(* IEC 61131-3 sources: Elmo_Master/Lasal_PRG/Elmo_EtherCAT_Test_4Axis/Class/LMCDiagnosticsService (part 2) *)

	if detailCode <> 0 then
		(pResponse + 12)^$UDINT := detailCode;
		RETURN;
	end_if;
	if ResponseCapacity < 156 then
		ResponseSize := -1;
		RETURN;
	end_if;

	_memset(dest:=pResponse, usByte:=0, cntr:=156);
	pResponse^$UINT := LMC_DIAG_SCHEMA_VERSION;
	(pResponse + 4)^$UINT := 0;
	(pResponse + 6)^$INT := 0;
	(pResponse + 8)^$UDINT := requestId;
	(pResponse + 12)^$UDINT := 0;
	(pResponse + 16)^$UINT := baseState$UINT;
	(pResponse + 18)^$UINT := EncoderMaintenanceState[recordBase + 1]$UINT;
	(pResponse + 20)^$UDINT := EncoderMaintenanceState[recordBase + 2]$UDINT;
	(pResponse + 24)^$UDINT := EncoderMaintenanceState[recordBase + 3]$UDINT;
	(pResponse + 28)^$UDINT := EncoderMaintenanceState[recordBase + 4]$UDINT;
	(pResponse + 32)^$UDINT := EncoderMaintenanceState[recordBase + 5]$UDINT;
	(pResponse + 36)^$UDINT := EncoderMaintenanceState[recordBase + 6]$UDINT;
	(pResponse + 40)^$UDINT := EncoderMaintenanceState[recordBase + 7]$UDINT;
	(pResponse + 44)^$UDINT := EncoderMaintenanceState[recordBase + 8]$UDINT;
	(pResponse + 48)^$UDINT := EncoderMaintenanceState[recordBase + 9]$UDINT;
	(pResponse + 52)^$UINT := EncoderMaintenanceState[recordBase + 10]$UINT;
	(pResponse + 54)^$UINT := EncoderMaintenanceState[recordBase + 11]$UINT;
	(pResponse + 56)^$UINT := EncoderMaintenanceState[recordBase + 12]$UINT;
	(pResponse + 58)^$UINT := 0;
	(pResponse + 60)^$UDINT := EncoderMaintenanceState[recordBase + 13]$UDINT;
	(pResponse + 64)^$UDINT := EncoderMaintenanceState[recordBase + 14]$UDINT;
	(pResponse + 68)^$UDINT := EncoderMaintenanceState[recordBase + 15]$UDINT;
	(pResponse + 72)^$UDINT := EncoderMaintenanceState[recordBase + 16]$UDINT;
	(pResponse + 76)^$UDINT := EncoderMaintenanceState[recordBase + 17]$UDINT;
	(pResponse + 80)^$UDINT := EncoderMaintenanceState[recordBase + 18]$UDINT;
	(pResponse + 84)^$UINT := EncoderMaintenanceState[recordBase + 19]$UINT;
	(pResponse + 86)^$INT := EncoderMaintenanceState[recordBase + 20]$INT;
	(pResponse + 88)^$UDINT := EncoderMaintenanceState[recordBase + 21]$UDINT;
	(pResponse + 92)^$UDINT := EncoderMaintenanceState[recordBase + 22]$UDINT;
	(pResponse + 96)^$UDINT := EncoderMaintenanceState[recordBase + 23]$UDINT;
	(pResponse + 100)^$UDINT := EncoderMaintenanceState[recordBase + 24]$UDINT;
	(pResponse + 104)^$UDINT := EncoderMaintenanceState[recordBase + 25]$UDINT;
	(pResponse + 108)^$UDINT := EncoderMaintenanceState[recordBase + 26]$UDINT;
	(pResponse + 112)^$UDINT := EncoderMaintenanceState[recordBase + 27]$UDINT;
	(pResponse + 116)^$UDINT := EncoderMaintenanceState[recordBase + 28]$UDINT;
	(pResponse + 120)^$UDINT := EncoderMaintenanceState[recordBase + 29]$UDINT;
	(pResponse + 124)^$UDINT := EncoderMaintenanceState[recordBase + 30]$UDINT;
	(pResponse + 128)^$UDINT := EncoderMaintenanceState[recordBase + 31]$UDINT;
	(pResponse + 132)^$UINT := EncoderMaintenanceState[recordBase + 32]$UINT;
	(pResponse + 134)^$UINT := 0;
	(pResponse + 136)^$DINT := EncoderMaintenanceState[recordBase + 33];
	(pResponse + 140)^$UDINT := EncoderMaintenanceState[recordBase + 34]$UDINT;
	(pResponse + 144)^$DINT := EncoderMaintenanceState[recordBase + 35];
	(pResponse + 148)^$UDINT := EncoderMaintenanceState[recordBase + 36]$UDINT;
	(pResponse + 152)^$UDINT := EncoderMaintenanceState[recordBase + 37]$UDINT;
	ResponseSize := 156;

END_FUNCTION

FUNCTION LMCDiagnosticsService::HandleEncoderMaintenanceRetire
	VAR_INPUT
		Reference 	: UINT;
		pRequest 	: ^USINT;
		pResponse 	: ^USINT;
		ResponseCapacity 	: UDINT;
		CallerSessionEpoch 	: UDINT;
		RequestSize 	: UDINT;
	END_VAR
	VAR_OUTPUT
		ResponseSize 	: DINT;
	END_VAR
	VAR
		driveReference : UINT;
		requestId, recordGeneration, detailCode : UDINT;
		rawState, baseState : UDINT;
		recordBase : DINT;
		stateValid : BOOL;
	END_VAR

	ResponseSize := -1;
	if (pResponse = NIL) | (ResponseCapacity < 16) then
		RETURN;
	end_if;
	_memset(dest:=pResponse, usByte:=0, cntr:=16);
	pResponse^$UINT := LMC_DIAG_SCHEMA_VERSION;
	(pResponse + 4)^$UINT := 1;
	(pResponse + 6)^$INT := LMC_DIAG_ERROR_ID;
	requestId := 0;
	if (pRequest <> NIL) & (RequestSize >= 8) then
		requestId := (pRequest + 4)^$UDINT;
	end_if;
	(pResponse + 8)^$UDINT := requestId;
	ResponseSize := 16;
	detailCode := LMC_DIAG_ENCODER_DETAIL_KEY_MISMATCH;

	if (pRequest = NIL) | (RequestSize <> 76) | (Reference <> 0) then
		(pResponse + 12)^$UDINT := detailCode;
		RETURN;
	end_if;
	driveReference := (pRequest + 44)^$UINT;
	recordGeneration := (pRequest + 72)^$UDINT;
	recordBase := 0;
	if (driveReference < 1) | (driveReference > 4) |
		(recordGeneration = 0) then
		(pResponse + 12)^$UDINT := detailCode;
		RETURN;
	end_if;

	recordBase := TO_DINT(driveReference - 1) *
		LMC_DIAG_ENCODER_RECORD_STRIDE;
	rawState := EncoderMaintenanceState[recordBase]$UDINT;
	baseState := rawState and 0x00007FFF;
	stateValid :=
		(rawState = LMC_DIAG_ENCODER_RECORD_SUCCEEDED) |
		(rawState = LMC_DIAG_ENCODER_RECORD_FAILED) |
		(rawState = LMC_DIAG_ENCODER_RECORD_ABORTED) |
		(rawState = (LMC_DIAG_ENCODER_RECORD_RETIRED OR
		 LMC_DIAG_ENCODER_RECORD_SUCCEEDED)) |
		(rawState = (LMC_DIAG_ENCODER_RECORD_RETIRED OR
		 LMC_DIAG_ENCODER_RECORD_FAILED)) |
		(rawState = (LMC_DIAG_ENCODER_RECORD_RETIRED OR
		 LMC_DIAG_ENCODER_RECORD_ABORTED));
	if rawState = 0 then
		detailCode := LMC_DIAG_ENCODER_DETAIL_NOT_FOUND;
	elsif rawState = LMC_DIAG_ENCODER_RECORD_RUNNING then
		detailCode := LMC_DIAG_ENCODER_DETAIL_INDETERMINATE;
	elsif stateValid = FALSE then
		detailCode := LMC_DIAG_ENCODER_DETAIL_STORE_CORRUPT;
	elsif EncoderMaintenanceState[recordBase + 36]$UDINT <>
		recordGeneration then
		detailCode := LMC_DIAG_ENCODER_DETAIL_KEY_MISMATCH;
	else
		ResponseSize := HandleEncoderMaintenanceOutcome(
			Reference:=Reference, pRequest:=pRequest,
			pResponse:=pResponse, ResponseCapacity:=ResponseCapacity,
			CallerSessionEpoch:=CallerSessionEpoch, RequestSize:=72);
		if (ResponseSize = 156) &
			((pResponse + 148)^$UDINT = recordGeneration) then
			if rawState = baseState then
				// State is the publication word. Setting the tombstone last makes
				// retrying the same exact retirement idempotent.
				EncoderMaintenanceState[recordBase] :=
					TO_DINT(baseState OR
					LMC_DIAG_ENCODER_RECORD_RETIRED);
			end_if;
			RETURN;
		end_if;
		detailCode := LMC_DIAG_ENCODER_DETAIL_KEY_MISMATCH;
	end_if;

	(pResponse + 4)^$UINT := 1;
	(pResponse + 6)^$INT := LMC_DIAG_ERROR_ID;
	(pResponse + 12)^$UDINT := detailCode;
	ResponseSize := 16;

END_FUNCTION

FUNCTION LMCDiagnosticsService::ProcessEncoderMaintenance
	VAR
		snapshot : ARRAY [0..303] OF USINT;
		preemptionSnapshot : ARRAY [0..215] OF USINT;
		completion : LMCSdoExecutor::LMCSdoExecutorResult;
		stage, recordBase, desiredTerminalState : DINT;
		axisReference, maintenanceObjectIndex : UINT;
		maintenanceSubIndex : USINT;
		maintenanceKind, preemptionCleanupKind : UINT;
		maintenanceWriteValue : UINT;
		axisMask, encoderProcessOperationToken, admissionToken, ownerGeneration : UDINT;
		callerSessionEpoch, requestSequence : UDINT;
		maintenanceCommandValue, timeoutMilliseconds : UDINT;
		expectedExecuteToken, safetyAdmissionToken, safetyOwnerGeneration : UDINT;
		serviceNow, serviceStartMs, cleanupStartMs : UDINT;
		elapsedMs, remainingMs, currentCycle, previousCycle : UDINT;
		healthOffset, valueOffset, controlWord, statusWord : UDINT;
		failureDetail, failureNative, verificationFlags : UDINT;
		axisError, actualPosition : DINT;
		copyResult, ownerResult, orphanResult, preemptionResult : DINT;
		startResult : iprStates;
		snapshotValid, newCycle, motorOff : BOOL;
		executorConnected, executorReusable, featureEnabled : BOOL;
		safeFailure, quarantine, preemptionSnapshotValid : BOOL;
		dispatchDefinitelyAbsent, publishPreemptionCleanup : BOOL;
	END_VAR

	stage := EncoderMaintenanceState[LMC_DIAG_ENCODER_RUNTIME_BASE];
	if stage = LMC_DIAG_ENCODER_STAGE_IDLE then
		RETURN;
	end_if;

	recordBase := EncoderMaintenanceState[154];
	axisReference := EncoderMaintenanceState[153]$UINT;
	admissionToken := EncoderMaintenanceState[160]$UDINT;
	ownerGeneration := EncoderMaintenanceState[161]$UDINT;
	_memset(dest:=#preemptionSnapshot[0], usByte:=0,
		cntr:=sizeof(preemptionSnapshot));
	preemptionResult := -1;
	if IsClientConnected(#AxisOwnership) & (admissionToken <> 0) &
		(ownerGeneration <> 0) then
		preemptionResult := AxisOwnership.CopyAxisOwnershipPreemption(
			PreemptedAdmissionToken:=admissionToken,
			PreemptedOwnerGeneration:=ownerGeneration,
			pDest:=#preemptionSnapshot[0],
			DestSize:=sizeof(preemptionSnapshot));
	end_if;
	if preemptionResult = LMC_DIAG_PREEMPT_PENDING_FREEZE then
		// Safety is only reserved. Freeze before changing any owner runtime word.
		RETURN;
	end_if;
	if (preemptionResult < 0) |
		(preemptionResult > LMC_DIAG_PREEMPT_CLEANUP_QUARANTINED) then
		EncoderMaintenanceState[179] :=
			LMC_DIAG_ENCODER_DETAIL_STORE_CORRUPT;
		EncoderMaintenanceState[180] := TO_DINT(0 - preemptionResult);
		EncoderMaintenanceState[152] :=
			LMC_DIAG_ENCODER_STAGE_QUARANTINED;
		RETURN;
	end_if;
	if (sizeof(EncoderMaintenanceState) <> 768) |
		(axisReference < 1) | (axisReference > 4) |
		(recordBase <> (TO_DINT(axisReference - 1) *
		 LMC_DIAG_ENCODER_RECORD_STRIDE)) |
		(EncoderMaintenanceState[recordBase] <>
		 LMC_DIAG_ENCODER_RECORD_RUNNING) then
		EncoderMaintenanceState[152] :=
			LMC_DIAG_ENCODER_STAGE_QUARANTINED;
		RETURN;
	end_if;

	axisMask := TO_UDINT(1) shl TO_UDINT(axisReference - 1);
	maintenanceKind := EncoderMaintenanceState[182]$UINT;
	maintenanceObjectIndex := EncoderMaintenanceState[157]$UINT;
	maintenanceSubIndex := EncoderMaintenanceState[158]$USINT;
	maintenanceCommandValue := EncoderMaintenanceState[159]$UDINT;
	maintenanceWriteValue := LMC_DIAG_ENCODER_RESET_VALUE;
	timeoutMilliseconds := EncoderMaintenanceState[recordBase + 14]$UDINT;
	encoderProcessOperationToken := EncoderMaintenanceState[155]$UDINT;
	callerSessionEpoch := EncoderMaintenanceState[162]$UDINT;
	requestSequence := EncoderMaintenanceState[163]$UDINT;
	serviceNow := ops.tAbsolute;
	serviceStartMs := EncoderMaintenanceState[164]$UDINT;
	cleanupStartMs := EncoderMaintenanceState[165]$UDINT;
	elapsedMs := serviceNow - serviceStartMs;
	previousCycle := EncoderMaintenanceState[166]$UDINT;
	currentCycle := previousCycle;
	controlWord := EncoderMaintenanceState[168]$UDINT;
	statusWord := EncoderMaintenanceState[169]$UDINT;
	axisError := EncoderMaintenanceState[170];
	actualPosition := EncoderMaintenanceState[171];
	expectedExecuteToken := 0;
	if maintenanceKind = 1 then
		expectedExecuteToken := 0x30325754;
	elsif maintenanceKind = 2 then
		expectedExecuteToken := 0x39315754;
	end_if;

	preemptionResult := HandleEncoderMaintenancePreemption(
		Stage:=stage,
		PreemptionResult:=preemptionResult,
		pPreemptionSnapshot:=#preemptionSnapshot[0],
		ServiceNow:=serviceNow);
	if preemptionResult <> 0 then
		RETURN;
	end_if;

	if stage = LMC_DIAG_ENCODER_STAGE_QUARANTINED then
		RETURN;
	end_if;
	EncoderMaintenanceServiceMilliseconds := serviceNow;

	snapshotValid := FALSE;
	newCycle := FALSE;
	motorOff := FALSE;
	copyResult := -1;
	if IsClientConnected(#InputLatch) then
		copyResult := InputLatch.CopySnapshot(
			pDest:=#snapshot[0], DestSize:=sizeof(snapshot));
	end_if;
	if (copyResult = 0) & (snapshot[0]$UDINT <> 0) then
		currentCycle := snapshot[0]$UDINT;
		healthOffset := 64 + TO_UDINT(axisReference - 1) * 36;
		valueOffset := 208 + TO_UDINT(axisReference - 1) * 24;
		controlWord := snapshot[TO_DINT(valueOffset + 8)]$UDINT;
		statusWord := snapshot[TO_DINT(valueOffset + 20)]$UDINT;
		axisError := snapshot[TO_DINT(healthOffset + 24)]$DINT;
		actualPosition := snapshot[TO_DINT(valueOffset + 12)]$DINT;
		snapshotValid :=
			(snapshot[12]$UDINT = 8) & (snapshot[16]$UDINT = 0) &
			((snapshot[40]$UDINT and 3) = 1) &
			(snapshot[TO_DINT(healthOffset)]$DINT <> 0) &
			(snapshot[TO_DINT(healthOffset + 4)]$UDINT = 8) &
			(snapshot[TO_DINT(healthOffset + 12)]$UDINT = 0) &
			(snapshot[TO_DINT(healthOffset + 16)]$UDINT <>
			 0xFFFFFFFF) &
			(snapshot[TO_DINT(healthOffset + 28)]$UDINT = currentCycle);
		newCycle := snapshotValid & (currentCycle <> previousCycle);
		motorOff := snapshotValid &
			((controlWord and 0x00000008) = 0) &
			((statusWord and 0x00000004) = 0);
		if snapshotValid then
			EncoderMaintenanceState[166] := currentCycle$DINT;
			EncoderMaintenanceState[168] := controlWord$DINT;
			EncoderMaintenanceState[169] := statusWord$DINT;
			EncoderMaintenanceState[170] := axisError;
			EncoderMaintenanceState[171] := actualPosition;
			EncoderMaintenanceState[recordBase + 32] := statusWord$DINT;
			EncoderMaintenanceState[recordBase + 33] := axisError;
			EncoderMaintenanceState[recordBase + 35] := actualPosition;
		end_if;
	end_if;

	executorConnected := FALSE;
	executorReusable := FALSE;
	case axisReference of
		1:
			executorConnected := IsClientConnected(#SdoAxis1) <> 0;
			if executorConnected then
				executorReusable := SdoAxis1.IsReusable();
			end_if;
		2:
			executorConnected := IsClientConnected(#SdoAxis2) <> 0;
			if executorConnected then
				executorReusable := SdoAxis2.IsReusable();
			end_if;
		3:
			executorConnected := IsClientConnected(#SdoAxis3) <> 0;
			if executorConnected then
				executorReusable := SdoAxis3.IsReusable();
			end_if;
		4:
			executorConnected := IsClientConnected(#SdoAxis4) <> 0;
			if executorConnected then
				executorReusable := SdoAxis4.IsReusable();
			end_if;
	end_case;

	featureEnabled :=
		((maintenanceKind = 1) &
		 (LMC_DIAG_ENCODER_TW20_ENABLED = TRUE)) |
		((maintenanceKind = 2) &
		 (LMC_DIAG_ENCODER_TW19_ENABLED = TRUE));
	safeFailure := FALSE;
	quarantine := FALSE;
	failureDetail := LMC_DIAG_ENCODER_DETAIL_EXECUTION;
	failureNative := 0;
	desiredTerminalState := LMC_DIAG_ENCODER_RECORD_FAILED;

	if (maintenanceObjectIndex <> 0x20FC) |
		(((maintenanceKind = 1) & (maintenanceSubIndex <> 0x02)) |
		 ((maintenanceKind = 2) & (maintenanceSubIndex <> 0x01))) |
		((maintenanceKind <> 1) & (maintenanceKind <> 2)) |
		(maintenanceCommandValue <> LMC_DIAG_ENCODER_RESET_VALUE) |
		(encoderProcessOperationToken = 0) | (admissionToken = 0) |
		(ownerGeneration = 0) | (callerSessionEpoch = 0) |
		(requestSequence = 0) | (timeoutMilliseconds < 1) |
		(timeoutMilliseconds > 60000) then
		quarantine := TRUE;
		failureNative := 17;
	elsif (featureEnabled = FALSE) &
		(stage <> LMC_DIAG_ENCODER_STAGE_RELEASE_OWNER) then
		if EncoderMaintenanceState[189]$UDINT = 0 then
			safeFailure := TRUE;
			failureDetail := LMC_DIAG_ENCODER_DETAIL_EXECUTION;
			failureNative := LMC_DIAG_ENCODER_DETAIL_COMPATIBILITY;
		else
			quarantine := TRUE;
			failureNative := LMC_DIAG_ENCODER_DETAIL_COMPATIBILITY;
		end_if;
	end_if;

	if (safeFailure = FALSE) & (quarantine = FALSE) then
		case stage of
			LMC_DIAG_ENCODER_STAGE_PRE_STABLE:
				if elapsedMs >= timeoutMilliseconds then
					safeFailure := TRUE;
					desiredTerminalState :=
						LMC_DIAG_ENCODER_RECORD_ABORTED;
					failureDetail := LMC_DIAG_ENCODER_DETAIL_ABORTED;
				elsif snapshotValid & (motorOff = FALSE) then
					safeFailure := TRUE;
					failureDetail := LMC_DIAG_ENCODER_DETAIL_SEMANTIC;
					failureNative := statusWord;
				elsif newCycle & motorOff then
					EncoderMaintenanceObservedLatchCycle := currentCycle;
					EncoderMaintenanceLatchAdvanceServiceMilliseconds :=
						serviceNow;
					EncoderMaintenanceLatchFreshSampleCount += 1;
					EncoderMaintenanceState[recordBase + 28] :=
						controlWord$DINT;
					EncoderMaintenanceState[recordBase + 30] :=
						statusWord$DINT;
					if EncoderMaintenanceLatchFreshSampleCount >= 3 then
						EncoderMaintenanceState[recordBase + 27]$UDINT :=
							EncoderMaintenanceState[recordBase + 27]$UDINT OR
							LMC_DIAG_ENCODER_VERIFY_MOTOR_OFF_PRE OR
							LMC_DIAG_ENCODER_VERIFY_NO_MOTION;
						EncoderMaintenanceState[152] :=
							LMC_DIAG_ENCODER_STAGE_DISPATCH;
					end_if;
				end_if;

			LMC_DIAG_ENCODER_STAGE_DISPATCH:
				if elapsedMs >= timeoutMilliseconds then
					safeFailure := TRUE;
					desiredTerminalState :=
						LMC_DIAG_ENCODER_RECORD_ABORTED;
					failureDetail := LMC_DIAG_ENCODER_DETAIL_ABORTED;
				elsif snapshotValid = FALSE then
					// Wait only within the same overall service-clock budget.
				elsif motorOff = FALSE then
					safeFailure := TRUE;
					failureDetail := LMC_DIAG_ENCODER_DETAIL_SEMANTIC;
					failureNative := statusWord;
				elsif (executorConnected = FALSE) | (executorReusable = FALSE) |
					(IsClientConnected(#AxisOwnership) = FALSE) then
					quarantine := TRUE;
					failureNative := 24;
				else
					ownerResult := AxisOwnership.ValidateAxisOwnership(
						CommandId:=0x7E53,
						Reference:=axisReference,
						ExpectedAxisMask:=axisMask,
						OwnerKind:=LMC_DIAG_OWNER_KIND_ENCODER,
						ResourceKind:=LMC_DIAG_RESOURCE_DIAGNOSTICS_SDO,
						AdmissionMode:=LMC_DIAG_ADMISSION_LIFECYCLE,
						CallerSessionEpoch:=callerSessionEpoch,
						RequestSequence:=requestSequence,
						AdmissionToken:=admissionToken,
						OwnerGeneration:=ownerGeneration,
						RequiredPhase:=LMC_DIAG_OWNER_PHASE_ACTIVE);
					if ownerResult <> 0 then
						quarantine := TRUE;
						failureNative := TO_UDINT(0 - ownerResult);
					elsif EncoderMaintenanceState[189]$UDINT <> 0 then
						// This is the irreversible one-shot dispatch claim. It is
						// never cleared for retry within an active record.
						quarantine := TRUE;
						failureNative := 25;
					else
						remainingMs := timeoutMilliseconds - elapsedMs;
						if remainingMs < 1 then
							remainingMs := 1;
						end_if;
						if remainingMs > 60000 then
							remainingMs := 60000;
						end_if;
						EncoderMaintenanceState[189]$UDINT := encoderProcessOperationToken;
						startResult := ERROR;
						case axisReference of
							1:
								startResult := SdoAxis1.TryStartWrite(
									OperationToken:=encoderProcessOperationToken,
									ObjectIndex:=maintenanceObjectIndex,
									SubIndex:=maintenanceSubIndex,
									pWriteData:=(#maintenanceWriteValue)$^USINT,
									WriteLength:=2, TimeoutMs:=remainingMs);
							2:
								startResult := SdoAxis2.TryStartWrite(
									OperationToken:=encoderProcessOperationToken,
									ObjectIndex:=maintenanceObjectIndex,
									SubIndex:=maintenanceSubIndex,
									pWriteData:=(#maintenanceWriteValue)$^USINT,
									WriteLength:=2, TimeoutMs:=remainingMs);
							3:
								startResult := SdoAxis3.TryStartWrite(
									OperationToken:=encoderProcessOperationToken,
									ObjectIndex:=maintenanceObjectIndex,
									SubIndex:=maintenanceSubIndex,
									pWriteData:=(#maintenanceWriteValue)$^USINT,
									WriteLength:=2, TimeoutMs:=remainingMs);
							4:
								startResult := SdoAxis4.TryStartWrite(
									OperationToken:=encoderProcessOperationToken,
									ObjectIndex:=maintenanceObjectIndex,
									SubIndex:=maintenanceSubIndex,
									pWriteData:=(#maintenanceWriteValue)$^USINT,
									WriteLength:=2, TimeoutMs:=remainingMs);
						end_case;
						if startResult = READY then
							EncoderMaintenanceState[156] := 1;
							EncoderMaintenanceState[152] :=
								LMC_DIAG_ENCODER_STAGE_WAIT_SDO;
							ownerResult := AxisOwnership.PublishAxisOwnership(
								AxisMask:=axisMask,
								AdmissionToken:=admissionToken,
								OwnerGeneration:=ownerGeneration,
								ReportKind:=LMC_DIAG_OWNER_REPORT_DISPATCH,
								ReportValue0:=TO_UDINT(maintenanceObjectIndex),
								ReportValue1:=encoderProcessOperationToken,
								ObservationCycle:=currentCycle);
							if ownerResult <> 0 then
								// Drain the accepted write before quarantine.
								EncoderMaintenanceState[176] := 1;
							end_if;
						else
							case axisReference of
								1: executorReusable := SdoAxis1.IsReusable();
								2: executorReusable := SdoAxis2.IsReusable();
								3: executorReusable := SdoAxis3.IsReusable();
								4: executorReusable := SdoAxis4.IsReusable();
							end_case;
							if executorReusable then
								safeFailure := TRUE;
								failureNative := TO_UDINT(startResult);
							else
								quarantine := TRUE;
								failureNative := TO_UDINT(startResult);
							end_if;
						end_if;
					end_if;
				end_if;

			LMC_DIAG_ENCODER_STAGE_WAIT_SDO:
				copyResult := -2;
				case axisReference of
					1: copyResult := SdoAxis1.CopyCompletion(
						ExpectedToken:=encoderProcessOperationToken,
						pDest:=#completion, DestSize:=sizeof(completion));
					2: copyResult := SdoAxis2.CopyCompletion(
						ExpectedToken:=encoderProcessOperationToken,
						pDest:=#completion, DestSize:=sizeof(completion));
					3: copyResult := SdoAxis3.CopyCompletion(
						ExpectedToken:=encoderProcessOperationToken,
						pDest:=#completion, DestSize:=sizeof(completion));
					4: copyResult := SdoAxis4.CopyCompletion(
						ExpectedToken:=encoderProcessOperationToken,
						pDest:=#completion, DestSize:=sizeof(completion));
				end_case;
				if copyResult = 0 then
					EncoderMaintenanceState[156] := 0;
					EncoderMaintenanceState[recordBase + 24] :=
						currentCycle$DINT;
					EncoderMaintenanceState[recordBase + 22] :=
						completion.AbortCode$DINT;
					EncoderMaintenanceState[recordBase + 27]$UDINT :=
						EncoderMaintenanceState[recordBase + 27]$UDINT OR
						LMC_DIAG_ENCODER_VERIFY_SDO_COMPLETE OR
						LMC_DIAG_ENCODER_VERIFY_EXECUTOR_DRAINED;
					case axisReference of
						1: executorReusable := SdoAxis1.IsReusable();
						2: executorReusable := SdoAxis2.IsReusable();
						3: executorReusable := SdoAxis3.IsReusable();
						4: executorReusable := SdoAxis4.IsReusable();
					end_case;
					if (completion.Token = encoderProcessOperationToken) &
						(completion.ValidationCode = 0) &
						(completion.OsResult = 0) &
						(completion.AbortCode = 0) &
						(completion.ObjectIndex = maintenanceObjectIndex) &
						(completion.SubIndex = maintenanceSubIndex) &
						(completion.IsWrite <> 0) &
						(completion.ActualLength = 2) &
						(completion.Reserved = 0) & executorReusable &
						(EncoderMaintenanceState[176] = 0) then
						EncoderMaintenanceLatchFreshSampleCount := 0;
						EncoderMaintenanceObservedLatchCycle := currentCycle;
						EncoderMaintenanceLatchAdvanceServiceMilliseconds :=
							serviceNow;
						EncoderMaintenanceState[152] :=
							LMC_DIAG_ENCODER_STAGE_POST_STABLE;
					else
						quarantine := TRUE;
						failureNative := completion.AbortCode;
						if failureNative = 0 then
							failureNative := TO_UDINT(0 - completion.OsResult);
						end_if;
					end_if;
				elsif copyResult <> -2 then
					quarantine := TRUE;
					failureNative := TO_UDINT(0 - copyResult);
				elsif elapsedMs >= timeoutMilliseconds then
					orphanResult := -1;
					case axisReference of
						1: orphanResult := SdoAxis1.MarkOrphan(
							ExpectedToken:=encoderProcessOperationToken);
						2: orphanResult := SdoAxis2.MarkOrphan(
							ExpectedToken:=encoderProcessOperationToken);
						3: orphanResult := SdoAxis3.MarkOrphan(
							ExpectedToken:=encoderProcessOperationToken);
						4: orphanResult := SdoAxis4.MarkOrphan(
							ExpectedToken:=encoderProcessOperationToken);
					end_case;
					if (orphanResult = 0) | (orphanResult = -2) then
						// -2 can mean RESULT_READY won the timeout race. The drain
						// stage consumes that exact completion before IsReusable.
						EncoderMaintenanceState[165] := serviceNow$DINT;
						EncoderMaintenanceState[177] := 1;
						EncoderMaintenanceState[152] :=
							LMC_DIAG_ENCODER_STAGE_DRAIN;
					else
						case axisReference of
							1: executorReusable := SdoAxis1.IsReusable();
							2: executorReusable := SdoAxis2.IsReusable();
							3: executorReusable := SdoAxis3.IsReusable();
							4: executorReusable := SdoAxis4.IsReusable();
						end_case;
						if executorReusable then
							quarantine := TRUE;
							failureNative := LMC_DIAG_ENCODER_DETAIL_ABORTED;
						end_if;
					end_if;
				end_if;

			LMC_DIAG_ENCODER_STAGE_POST_STABLE:
				if elapsedMs >= timeoutMilliseconds then
					quarantine := TRUE;
					failureNative := LMC_DIAG_ENCODER_DETAIL_ABORTED;
				elsif executorReusable = FALSE then
					quarantine := TRUE;
					failureNative := 24;
				elsif snapshotValid & (motorOff = FALSE) then
					quarantine := TRUE;
					failureDetail := LMC_DIAG_ENCODER_DETAIL_SEMANTIC;
					failureNative := statusWord;
				elsif newCycle & motorOff then
					EncoderMaintenanceObservedLatchCycle := currentCycle;
					EncoderMaintenanceLatchAdvanceServiceMilliseconds :=
						serviceNow;
					EncoderMaintenanceLatchFreshSampleCount += 1;
					EncoderMaintenanceState[recordBase + 29] :=
						controlWord$DINT;
					EncoderMaintenanceState[recordBase + 31] :=
						statusWord$DINT;
					if EncoderMaintenanceLatchFreshSampleCount >= 3 then
						EncoderMaintenanceState[recordBase + 27]$UDINT :=
							EncoderMaintenanceState[recordBase + 27]$UDINT OR
							LMC_DIAG_ENCODER_VERIFY_MOTOR_OFF_POST OR
							LMC_DIAG_ENCODER_VERIFY_STABLE_WINDOW OR
							LMC_DIAG_ENCODER_VERIFY_POST_WRITE_STATE OR
							LMC_DIAG_ENCODER_VERIFY_NO_MOTION;
						EncoderMaintenanceState[178] :=
							LMC_DIAG_ENCODER_RECORD_SUCCEEDED;
						EncoderMaintenanceState[152] :=
							LMC_DIAG_ENCODER_STAGE_RELEASE_OWNER;
					end_if;
				end_if;

			LMC_DIAG_ENCODER_STAGE_RELEASE_OWNER:
				desiredTerminalState := EncoderMaintenanceState[178];
				if IsClientConnected(#AxisOwnership) = FALSE then
					quarantine := TRUE;
					failureNative := 24;
				elsif desiredTerminalState =
					LMC_DIAG_ENCODER_RECORD_SUCCEEDED then
					verificationFlags :=
						EncoderMaintenanceState[recordBase + 27]$UDINT;
					if verificationFlags <>
						(LMC_DIAG_ENCODER_VERIFY_ALL and
						 NOT(LMC_DIAG_ENCODER_VERIFY_OWNER_CLEANUP)) then
						quarantine := TRUE;
						failureNative := verificationFlags;
					else
						ownerResult := AxisOwnership.PublishAxisOwnership(
							AxisMask:=axisMask,
							AdmissionToken:=admissionToken,
							OwnerGeneration:=ownerGeneration,
							ReportKind:=
								LMC_DIAG_OWNER_REPORT_TERMINAL_SUCCESS,
							ReportValue0:=0,
							ReportValue1:=verificationFlags,
							ObservationCycle:=currentCycle);
						if ownerResult = 0 then
							EncoderMaintenanceState[recordBase + 27]$UDINT :=
								LMC_DIAG_ENCODER_VERIFY_ALL;
							EncoderMaintenanceState[recordBase + 19] := 0;
							EncoderMaintenanceState[recordBase + 20] := 0;
							EncoderMaintenanceState[recordBase + 21] := 0;
							EncoderMaintenanceState[recordBase + 22] := 0;
							EncoderMaintenanceState[recordBase + 25] :=
								currentCycle$DINT;
							EncoderMaintenanceState[recordBase + 26] := 0;
							// Terminal state is the final publication word, after the
							// executor is reusable and the owner release succeeded.
							EncoderMaintenanceState[recordBase] :=
								LMC_DIAG_ENCODER_RECORD_SUCCEEDED;
							_memset(
								dest:=#EncoderMaintenanceState[152],
								usByte:=0, cntr:=34 * 4);
							EncoderMaintenanceServiceMilliseconds := 0;
							EncoderMaintenanceObservedLatchCycle := 0;
							EncoderMaintenanceLatchAdvanceServiceMilliseconds := 0;
							EncoderMaintenanceLatchFreshSampleCount := 0;
							RETURN;
						else
							quarantine := TRUE;
							failureNative := TO_UDINT(0 - ownerResult);
						end_if;
					end_if;
				elsif (desiredTerminalState =
					LMC_DIAG_ENCODER_RECORD_FAILED) |
					(desiredTerminalState =
					 LMC_DIAG_ENCODER_RECORD_ABORTED) then
					ownerResult := AxisOwnership.PublishAxisOwnership(
						AxisMask:=axisMask,
						AdmissionToken:=admissionToken,
						OwnerGeneration:=ownerGeneration,
						ReportKind:=
							LMC_DIAG_OWNER_REPORT_TERMINAL_SAFE_FAILURE,
						ReportValue0:=EncoderMaintenanceState[179]$UDINT,
						ReportValue1:=EncoderMaintenanceState[180]$UDINT,
						ObservationCycle:=currentCycle);
					if ownerResult = 0 then
						EncoderMaintenanceState[recordBase + 27]$UDINT :=
							EncoderMaintenanceState[recordBase + 27]$UDINT OR
							LMC_DIAG_ENCODER_VERIFY_OWNER_CLEANUP;
						EncoderMaintenanceState[recordBase + 19] := 1;
						EncoderMaintenanceState[recordBase + 20] :=
							LMC_DIAG_ERROR_ID;
						EncoderMaintenanceState[recordBase + 21] :=
							EncoderMaintenanceState[179];
						EncoderMaintenanceState[recordBase + 22] := 0;
						EncoderMaintenanceState[recordBase + 25] :=
							currentCycle$DINT;
						EncoderMaintenanceState[recordBase + 26] := 0;
						EncoderMaintenanceState[recordBase] :=
							desiredTerminalState;
						_memset(dest:=#EncoderMaintenanceState[152],
							usByte:=0, cntr:=34 * 4);
						EncoderMaintenanceServiceMilliseconds := 0;
						EncoderMaintenanceObservedLatchCycle := 0;
						EncoderMaintenanceLatchAdvanceServiceMilliseconds := 0;
						EncoderMaintenanceLatchFreshSampleCount := 0;
						RETURN;
					else
						quarantine := TRUE;
						failureNative := TO_UDINT(0 - ownerResult);
					end_if;
				else
					quarantine := TRUE;
					failureNative := 17;
				end_if;

			LMC_DIAG_ENCODER_STAGE_DRAIN:
				copyResult := -2;
				case axisReference of
					1: copyResult := SdoAxis1.CopyCompletion(
						ExpectedToken:=encoderProcessOperationToken,
						pDest:=#completion, DestSize:=sizeof(completion));
					2: copyResult := SdoAxis2.CopyCompletion(
						ExpectedToken:=encoderProcessOperationToken,
						pDest:=#completion, DestSize:=sizeof(completion));
					3: copyResult := SdoAxis3.CopyCompletion(
						ExpectedToken:=encoderProcessOperationToken,
						pDest:=#completion, DestSize:=sizeof(completion));
					4: copyResult := SdoAxis4.CopyCompletion(
						ExpectedToken:=encoderProcessOperationToken,
						pDest:=#completion, DestSize:=sizeof(completion));
				end_case;
				if copyResult = 0 then
					EncoderMaintenanceState[156] := 0;
				end_if;
				case axisReference of
					1: executorReusable := SdoAxis1.IsReusable();
					2: executorReusable := SdoAxis2.IsReusable();
					3: executorReusable := SdoAxis3.IsReusable();
					4: executorReusable := SdoAxis4.IsReusable();
				end_case;
				if (copyResult <> 0) & (copyResult <> -2) &
					(executorReusable = FALSE) then
					quarantine := TRUE;
					failureDetail := LMC_DIAG_ENCODER_DETAIL_ABORTED;
					failureNative := TO_UDINT(0 - copyResult);
				elsif executorReusable then
					// The late callback drained, but the write may have occurred.
					// Retaining owner quarantine is safer than a false terminal.
					quarantine := TRUE;
					failureDetail := LMC_DIAG_ENCODER_DETAIL_ABORTED;
					failureNative := LMC_DIAG_ENCODER_DETAIL_ABORTED;
				elsif (cleanupStartMs <> 0) &
					((serviceNow - cleanupStartMs) > 1000) then
					quarantine := TRUE;
					failureDetail := LMC_DIAG_ENCODER_DETAIL_ABORTED;
					failureNative := LMC_DIAG_ENCODER_DETAIL_ABORTED;
				end_if;

		else
			quarantine := TRUE;
			failureNative := 17;
		end_case;
	end_if;

	if safeFailure then
		EncoderMaintenanceState[178] := desiredTerminalState;
		EncoderMaintenanceState[179] := failureDetail$DINT;
		EncoderMaintenanceState[180] := failureNative$DINT;
		EncoderMaintenanceState[152] :=
			LMC_DIAG_ENCODER_STAGE_RELEASE_OWNER;
		RETURN;
	end_if;

	if quarantine then
		EncoderMaintenanceState[179] := failureDetail$DINT;
		EncoderMaintenanceState[180] := failureNative$DINT;
		EncoderMaintenanceState[152] :=
			LMC_DIAG_ENCODER_STAGE_QUARANTINED;
		ownerResult := -1;
		if IsClientConnected(#AxisOwnership) &
			(admissionToken <> 0) & (ownerGeneration <> 0) then
			ownerResult := AxisOwnership.PublishAxisOwnership(
				AxisMask:=axisMask,
				AdmissionToken:=admissionToken,
				OwnerGeneration:=ownerGeneration,
				ReportKind:=LMC_DIAG_OWNER_REPORT_QUARANTINE,
				ReportValue0:=failureDetail,
				ReportValue1:=failureNative,
				ObservationCycle:=currentCycle);
			if ownerResult <> 0 then
				EncoderMaintenanceState[190] := ownerResult;
				EncoderMaintenanceState[191] := 1;
			end_if;
		else
			EncoderMaintenanceState[190] := ownerResult;
			EncoderMaintenanceState[191] := 1;
		end_if;
	end_if;

END_FUNCTION

FUNCTION LMCDiagnosticsService::HandleEncoderMaintenancePreemption
	VAR_INPUT
		Stage 	: DINT;
		PreemptionResult 	: DINT;
		pPreemptionSnapshot 	: ^USINT;
		ServiceNow 	: UDINT;
	END_VAR
	VAR_OUTPUT
		Result 	: DINT;
	END_VAR
	VAR
		completion : LMCSdoExecutor::LMCSdoExecutorResult;
		recordBase : DINT;
		axisReference, maintenanceObjectIndex : UINT;
		maintenanceSubIndex : USINT;
		maintenanceKind, preemptionCleanupKind : UINT;
		axisMask, encoderProcessOperationToken : UDINT;
		admissionToken, ownerGeneration : UDINT;
		callerSessionEpoch, requestSequence : UDINT;
		maintenanceCommandValue, timeoutMilliseconds : UDINT;
		expectedExecuteToken, safetyAdmissionToken : UDINT;
		safetyOwnerGeneration, cleanupStartMs : UDINT;
		currentCycle, previousCycle : UDINT;
		copyResult, ownerResult, orphanResult : DINT;
		executorConnected, executorReusable : BOOL;
		preemptionSnapshotValid, dispatchDefinitelyAbsent : BOOL;
		publishPreemptionCleanup : BOOL;
	END_VAR

	Result := 1;
	recordBase := EncoderMaintenanceState[154];
	axisReference := EncoderMaintenanceState[153]$UINT;
	admissionToken := EncoderMaintenanceState[160]$UDINT;
	ownerGeneration := EncoderMaintenanceState[161]$UDINT;
	axisMask := TO_UDINT(1) shl TO_UDINT(axisReference - 1);
	maintenanceKind := EncoderMaintenanceState[182]$UINT;
	maintenanceObjectIndex := EncoderMaintenanceState[157]$UINT;
	maintenanceSubIndex := EncoderMaintenanceState[158]$USINT;
	maintenanceCommandValue := EncoderMaintenanceState[159]$UDINT;
	timeoutMilliseconds := EncoderMaintenanceState[recordBase + 14]$UDINT;
	encoderProcessOperationToken := EncoderMaintenanceState[155]$UDINT;
	callerSessionEpoch := EncoderMaintenanceState[162]$UDINT;
	requestSequence := EncoderMaintenanceState[163]$UDINT;
	cleanupStartMs := EncoderMaintenanceState[165]$UDINT;
	previousCycle := EncoderMaintenanceState[166]$UDINT;
	currentCycle := previousCycle;
	expectedExecuteToken := 0;
	if maintenanceKind = 1 then
		expectedExecuteToken := 0x30325754;
	elsif maintenanceKind = 2 then
		expectedExecuteToken := 0x39315754;
	end_if;

	if preemptionResult <> 0 then
		preemptionSnapshotValid :=
			((pPreemptionSnapshot + 0)^$UDINT =
			 LMC_DIAG_PREEMPT_SNAPSHOT_MAGIC) &
			((pPreemptionSnapshot + 4)^$UDINT =
			 LMC_DIAG_PREEMPT_SNAPSHOT_VERSION) &
			((pPreemptionSnapshot + 8)^$UDINT =
			 LMC_DIAG_PREEMPT_SNAPSHOT_HEADER_SIZE) &
			((pPreemptionSnapshot + 12)^$UDINT =
			 LMC_DIAG_PREEMPT_SNAPSHOT_TOTAL_SIZE) &
			((pPreemptionSnapshot + 16)^$DINT = preemptionResult) &
			((pPreemptionSnapshot + 32)^$UDINT = axisMask) &
			((pPreemptionSnapshot + 36)^$UDINT = admissionToken) &
			((pPreemptionSnapshot + 40)^$UDINT = ownerGeneration) &
			((pPreemptionSnapshot + 44)^$UDINT = callerSessionEpoch) &
			((pPreemptionSnapshot + 48)^$UDINT = requestSequence) &
			((pPreemptionSnapshot + 52)^$UDINT = 0x7E53) &
			((pPreemptionSnapshot + 56)^$UDINT = TO_UDINT(axisReference)) &
			((pPreemptionSnapshot + 60)^$UDINT = LMC_DIAG_OWNER_KIND_ENCODER) &
			((pPreemptionSnapshot + 64)^$UDINT =
			 LMC_DIAG_RESOURCE_DIAGNOSTICS_SDO) &
			((pPreemptionSnapshot + 68)^$UDINT =
			 LMC_DIAG_ADMISSION_LIFECYCLE) &
			(encoderProcessOperationToken <> 0) &
			(callerSessionEpoch <> 0) & (requestSequence <> 0) &
			(maintenanceObjectIndex = 0x20FC) &
			(((maintenanceKind = 1) & (maintenanceSubIndex = 0x02)) |
			 ((maintenanceKind = 2) & (maintenanceSubIndex = 0x01))) &
			((EncoderMaintenanceState[156] = 0) |
			 (EncoderMaintenanceState[156] = 1)) &
			((EncoderMaintenanceState[189]$UDINT = 0) |
			 (EncoderMaintenanceState[189]$UDINT =
			  encoderProcessOperationToken)) &
			((pPreemptionSnapshot + 72)^$UDINT >=
			 LMC_DIAG_OWNER_STATE_TW20_QUEUED) &
			((pPreemptionSnapshot + 72)^$UDINT <=
			 LMC_DIAG_OWNER_STATE_TW20_DRAINING) &
			((pPreemptionSnapshot + 76)^$UDINT = 72) &
			(((pPreemptionSnapshot + 104)^$UDINT and axisMask) = axisMask) &
			((pPreemptionSnapshot + 108)^$UDINT <> 0) &
			((pPreemptionSnapshot + 112)^$UDINT <> 0) &
			(((pPreemptionSnapshot + 124)^$UDINT =
			  LMC_DIAG_OWNER_STATE_SAFETY_PREEMPTING) |
			 ((pPreemptionSnapshot + 124)^$UDINT =
			  LMC_DIAG_OWNER_STATE_QUARANTINED)) &
			((pPreemptionSnapshot + 136)^$UDINT =
			 LMC_DIAG_ADMISSION_SAFETY) &
			((pPreemptionSnapshot + 144)^$UINT = LMC_DIAG_SCHEMA_VERSION) &
			((pPreemptionSnapshot + 146)^$UINT = 0) &
			((pPreemptionSnapshot + 148)^$UDINT =
			 EncoderMaintenanceState[recordBase + 5]$UDINT) &
			((pPreemptionSnapshot + 152)^$UDINT =
			 EncoderMaintenanceState[recordBase + 2]$UDINT) &
			((pPreemptionSnapshot + 156)^$UDINT =
			 EncoderMaintenanceState[recordBase + 3]$UDINT) &
			((pPreemptionSnapshot + 160)^$UDINT =
			 EncoderMaintenanceState[recordBase + 4]$UDINT) &
			((pPreemptionSnapshot + 164)^$UDINT =
			 EncoderMaintenanceState[recordBase + 6]$UDINT) &
			((pPreemptionSnapshot + 168)^$UDINT =
			 EncoderMaintenanceState[recordBase + 7]$UDINT) &
			((pPreemptionSnapshot + 172)^$UDINT =
			 EncoderMaintenanceState[recordBase + 8]$UDINT) &
			((pPreemptionSnapshot + 176)^$UDINT =
			 EncoderMaintenanceState[recordBase + 9]$UDINT) &
			((pPreemptionSnapshot + 180)^$UINT = maintenanceKind) &
			((pPreemptionSnapshot + 182)^$UINT =
			 EncoderMaintenanceState[recordBase + 10]$UINT) &
			((pPreemptionSnapshot + 184)^$UINT = axisReference) &
			((pPreemptionSnapshot + 186)^$UINT =
			 EncoderMaintenanceState[recordBase + 12]$UINT) &
			((pPreemptionSnapshot + 188)^$UDINT = maintenanceCommandValue) &
			((pPreemptionSnapshot + 192)^$UDINT = timeoutMilliseconds) &
			((pPreemptionSnapshot + 196)^$UDINT =
			 EncoderMaintenanceState[recordBase + 15]$UDINT) &
			((pPreemptionSnapshot + 200)^$UDINT =
			 EncoderMaintenanceState[recordBase + 16]$UDINT) &
			((pPreemptionSnapshot + 204)^$UDINT =
			 EncoderMaintenanceState[recordBase + 17]$UDINT) &
			((pPreemptionSnapshot + 208)^$UDINT =
			 EncoderMaintenanceState[recordBase + 18]$UDINT) &
			((pPreemptionSnapshot + 212)^$UDINT = expectedExecuteToken);
		if preemptionResult = LMC_DIAG_PREEMPT_CLEANUP_REQUIRED then
			preemptionSnapshotValid := preemptionSnapshotValid &
				(((pPreemptionSnapshot + 24)^$UDINT and axisMask) = axisMask) &
				(((pPreemptionSnapshot + 28)^$UDINT and axisMask) = 0) &
				((pPreemptionSnapshot + 124)^$UDINT <>
				 LMC_DIAG_OWNER_STATE_RESERVED);
		elsif preemptionResult = LMC_DIAG_PREEMPT_CLEANUP_COMPLETE then
			preemptionSnapshotValid := preemptionSnapshotValid &
				(((pPreemptionSnapshot + 28)^$UDINT and axisMask) = axisMask);
		end_if;
		if preemptionSnapshotValid = FALSE then
			EncoderMaintenanceState[179] :=
				LMC_DIAG_ENCODER_DETAIL_STORE_CORRUPT;
			EncoderMaintenanceState[180] := 43;
			EncoderMaintenanceState[152] :=
				LMC_DIAG_ENCODER_STAGE_QUARANTINED;
			RETURN;
		end_if;

		if preemptionResult = LMC_DIAG_PREEMPT_CLEANUP_COMPLETE then
			EncoderMaintenanceState[recordBase + 27]$UDINT :=
				EncoderMaintenanceState[recordBase + 27]$UDINT OR
				LMC_DIAG_ENCODER_VERIFY_OWNER_CLEANUP;
			EncoderMaintenanceState[recordBase + 19] := 1;
			EncoderMaintenanceState[recordBase + 20] := LMC_DIAG_ERROR_ID;
			EncoderMaintenanceState[recordBase + 21] :=
				LMC_DIAG_ENCODER_DETAIL_ABORTED;
			EncoderMaintenanceState[recordBase + 22] := 0;
			EncoderMaintenanceState[recordBase + 25] := currentCycle$DINT;
			EncoderMaintenanceState[recordBase + 26] := 0;
			EncoderMaintenanceState[recordBase] :=
				LMC_DIAG_ENCODER_RECORD_ABORTED;
			_memset(dest:=#EncoderMaintenanceState[152], usByte:=0,
				cntr:=34 * 4);
			EncoderMaintenanceServiceMilliseconds := 0;
			EncoderMaintenanceObservedLatchCycle := 0;
			EncoderMaintenanceLatchAdvanceServiceMilliseconds := 0;
			EncoderMaintenanceLatchFreshSampleCount := 0;
			RETURN;
		elsif preemptionResult =
			LMC_DIAG_PREEMPT_CLEANUP_QUARANTINED then
			EncoderMaintenanceState[179] :=
				LMC_DIAG_ENCODER_DETAIL_ABORTED;
			EncoderMaintenanceState[180] :=
				LMC_DIAG_ENCODER_DETAIL_INDETERMINATE;
			EncoderMaintenanceState[152] :=
				LMC_DIAG_ENCODER_STAGE_QUARANTINED;
			RETURN;
		end_if;

		// CLEANUP_REQUIRED is authorized only by this immutable coordinator
		// snapshot. Never use the preempted token for ordinary publication.
		safetyAdmissionToken := (pPreemptionSnapshot + 108)^$UDINT;
		safetyOwnerGeneration := (pPreemptionSnapshot + 112)^$UDINT;
		dispatchDefinitelyAbsent :=
			(EncoderMaintenanceState[189]$UDINT = 0) &
			(EncoderMaintenanceState[156] = 0) &
			((stage = LMC_DIAG_ENCODER_STAGE_PRE_STABLE) |
			 (stage = LMC_DIAG_ENCODER_STAGE_DISPATCH) |
			 (stage = LMC_DIAG_ENCODER_STAGE_RELEASE_OWNER)) &
			((pPreemptionSnapshot + 72)^$UDINT =
			 LMC_DIAG_OWNER_STATE_TW20_QUEUED);
		if dispatchDefinitelyAbsent then
			ownerResult := AxisOwnership.PublishAxisOwnershipPreemptionCleanup(
				ExpectedAxisMask:=axisMask,
				PreemptedAdmissionToken:=admissionToken,
				PreemptedOwnerGeneration:=ownerGeneration,
				SafetyAdmissionToken:=safetyAdmissionToken,
				SafetyOwnerGeneration:=safetyOwnerGeneration,
				CleanupKind:=LMC_DIAG_PREEMPT_CLEANUP_SAFE,
				ReportValue0:=LMC_DIAG_ENCODER_DETAIL_ABORTED,
				ReportValue1:=0,
				ObservationCycle:=currentCycle);
			if (ownerResult = 0) | (ownerResult = 1) then
				EncoderMaintenanceState[recordBase + 27]$UDINT :=
					EncoderMaintenanceState[recordBase + 27]$UDINT OR
					LMC_DIAG_ENCODER_VERIFY_OWNER_CLEANUP;
				EncoderMaintenanceState[recordBase + 19] := 1;
				EncoderMaintenanceState[recordBase + 20] := LMC_DIAG_ERROR_ID;
				EncoderMaintenanceState[recordBase + 21] :=
					LMC_DIAG_ENCODER_DETAIL_ABORTED;
				EncoderMaintenanceState[recordBase + 22] := 0;
				EncoderMaintenanceState[recordBase + 25] := currentCycle$DINT;
				EncoderMaintenanceState[recordBase + 26] := 0;
				EncoderMaintenanceState[recordBase] :=
					LMC_DIAG_ENCODER_RECORD_ABORTED;
				_memset(dest:=#EncoderMaintenanceState[152], usByte:=0,
					cntr:=34 * 4);
				EncoderMaintenanceServiceMilliseconds := 0;
				EncoderMaintenanceObservedLatchCycle := 0;
				EncoderMaintenanceLatchAdvanceServiceMilliseconds := 0;
				EncoderMaintenanceLatchFreshSampleCount := 0;
			else
				EncoderMaintenanceState[190] := ownerResult;
				EncoderMaintenanceState[179] :=
					LMC_DIAG_ENCODER_DETAIL_ABORTED;
				EncoderMaintenanceState[180] := TO_DINT(0 - ownerResult);
				EncoderMaintenanceState[191] := 1;
				EncoderMaintenanceState[152] :=
					LMC_DIAG_ENCODER_STAGE_QUARANTINED;
				RETURN;
			end_if;
			RETURN;
		end_if;

		// The irreversible dispatch claim means the write may have occurred.
		// Drain the exact token and require executor reuse before quarantine.
		if cleanupStartMs = 0 then
			cleanupStartMs := serviceNow;
			EncoderMaintenanceState[165] := cleanupStartMs$DINT;
		end_if;
		EncoderMaintenanceState[177] := 1;
		EncoderMaintenanceState[152] := LMC_DIAG_ENCODER_STAGE_DRAIN;
		executorConnected := FALSE;
		executorReusable := FALSE;
		case axisReference of
			1: executorConnected := IsClientConnected(#SdoAxis1) <> 0;
			2: executorConnected := IsClientConnected(#SdoAxis2) <> 0;
			3: executorConnected := IsClientConnected(#SdoAxis3) <> 0;
			4: executorConnected := IsClientConnected(#SdoAxis4) <> 0;
		end_case;
		copyResult := -2;
		if executorConnected then
			case axisReference of
				1: copyResult := SdoAxis1.CopyCompletion(
					ExpectedToken:=encoderProcessOperationToken,
					pDest:=#completion, DestSize:=sizeof(completion));
				2: copyResult := SdoAxis2.CopyCompletion(
					ExpectedToken:=encoderProcessOperationToken,
					pDest:=#completion, DestSize:=sizeof(completion));
				3: copyResult := SdoAxis3.CopyCompletion(
					ExpectedToken:=encoderProcessOperationToken,
					pDest:=#completion, DestSize:=sizeof(completion));
				4: copyResult := SdoAxis4.CopyCompletion(
					ExpectedToken:=encoderProcessOperationToken,
					pDest:=#completion, DestSize:=sizeof(completion));
			end_case;
			if copyResult = 0 then
				EncoderMaintenanceState[156] := 0;
				// Exact completion consumption proves this token is retired.
				EncoderMaintenanceState[181] := 1;
			elsif copyResult = -2 then
				orphanResult := -1;
				case axisReference of
					1: orphanResult := SdoAxis1.MarkOrphan(
						ExpectedToken:=encoderProcessOperationToken);
					2: orphanResult := SdoAxis2.MarkOrphan(
						ExpectedToken:=encoderProcessOperationToken);
					3: orphanResult := SdoAxis3.MarkOrphan(
						ExpectedToken:=encoderProcessOperationToken);
					4: orphanResult := SdoAxis4.MarkOrphan(
						ExpectedToken:=encoderProcessOperationToken);
				end_case;
				if (orphanResult = 0) | (orphanResult = -2) then
					// IsReusable below supplies the matching drain proof.
					EncoderMaintenanceState[181] := 1;
				end_if;
			end_if;
			case axisReference of
				1: executorReusable := SdoAxis1.IsReusable();
				2: executorReusable := SdoAxis2.IsReusable();
				3: executorReusable := SdoAxis3.IsReusable();
				4: executorReusable := SdoAxis4.IsReusable();
			end_case;
		end_if;
		publishPreemptionCleanup := executorReusable |
			(executorConnected = FALSE) |
			(copyResult < -2) |
			((serviceNow - cleanupStartMs) > 1000);
		if publishPreemptionCleanup = FALSE then
			RETURN;
		end_if;
		if executorReusable & (EncoderMaintenanceState[181] <> 0) then
			preemptionCleanupKind :=
				LMC_DIAG_PREEMPT_CLEANUP_COMPLETE_QUARANTINE;
		else
			preemptionCleanupKind :=
				LMC_DIAG_PREEMPT_CLEANUP_INCOMPLETE_QUARANTINE;
		end_if;
		ownerResult := AxisOwnership.PublishAxisOwnershipPreemptionCleanup(
			ExpectedAxisMask:=axisMask,
			PreemptedAdmissionToken:=admissionToken,
			PreemptedOwnerGeneration:=ownerGeneration,
			SafetyAdmissionToken:=safetyAdmissionToken,
			SafetyOwnerGeneration:=safetyOwnerGeneration,
			CleanupKind:=preemptionCleanupKind,
			ReportValue0:=encoderProcessOperationToken,
			ReportValue1:=TO_UDINT(copyResult),
			ObservationCycle:=currentCycle);
		if (ownerResult <> 0) & (ownerResult <> 1) then
			EncoderMaintenanceState[190] := ownerResult;
			EncoderMaintenanceState[179] :=
				LMC_DIAG_ENCODER_DETAIL_ABORTED;
			EncoderMaintenanceState[180] := TO_DINT(0 - ownerResult);
			EncoderMaintenanceState[191] := 1;
			EncoderMaintenanceState[152] :=
				LMC_DIAG_ENCODER_STAGE_QUARANTINED;
			RETURN;
		end_if;
		EncoderMaintenanceState[179] :=
			LMC_DIAG_ENCODER_DETAIL_ABORTED;
		EncoderMaintenanceState[180] := TO_DINT(copyResult);
		EncoderMaintenanceState[152] :=
			LMC_DIAG_ENCODER_STAGE_QUARANTINED;
		RETURN;
	end_if;
	Result := 0;

END_FUNCTION

FUNCTION LMCDiagnosticsService::HandleAxisDs402HomeStart
	VAR_INPUT
		Reference 	: UINT;
		pRequest 	: ^USINT;
		pResponse 	: ^USINT;
		ResponseCapacity 	: UDINT;
		CallerSessionEpoch 	: UDINT;
		RequestSequence 	: UDINT;
		AdmissionToken 	: UDINT;
		OwnerGeneration 	: UDINT;
		RequestSize 	: UDINT;
	END_VAR
	VAR_OUTPUT
		ResponseSize 	: DINT;
	END_VAR
	VAR
		schemaVersion, requestFlags : UINT;
		homingMethod, homePosition, velocity, acceleration : DINT;
		distanceLimit, torqueLimit : DINT;
		bufferMode, reservedValue : UINT;
		requestId, diagnosticsBuild, bootId, mapRevision : UDINT;
		intent0, intent1, intent2, intent3 : UDINT;
		timeoutMs, executeToken, currentBootId, detailCode : UDINT;
		nextGeneration, currentCycle, serviceStart, healthOffset, valueOffset : UDINT;
		axisMask : UDINT;
		rawStartState, baseStartState : UDINT;
		statusWord : UDINT;
		recordBase : DINT;
		copyResult, ownerResult, rollbackResult : DINT;
		intentBodyCompareResult, intentTailCompareResult : UDINT;
		snapshot : ARRAY [0..303] OF USINT;
		executorConnected, executorReusable : BOOL;
		journalEligible, journalPrepared, preflightOnly : BOOL;
		intentMatches : BOOL;
	END_VAR

	ResponseSize := -1;
	if (pResponse = NIL) | (ResponseCapacity < 24) then
		RETURN;
	end_if;

	_memset(dest:=pResponse, usByte:=0, cntr:=24);
	pResponse^$UINT := LMC_DIAG_SCHEMA_VERSION;
	(pResponse + 4)^$UINT := 1;
	(pResponse + 6)^$INT := LMC_DIAG_ADMIN_ERROR_ID;
	detailCode := 9;
	requestId := 0;
	homingMethod := 0;
	if (pRequest <> NIL) & (RequestSize >= 8) then
		requestId := (pRequest + 4)^$UDINT;
	end_if;
	if (pRequest <> NIL) & (RequestSize >= 40) then
		homingMethod := (pRequest + 36)^$DINT;
	end_if;
	(pResponse + 8)^$UDINT := requestId;
	(pResponse + 16)^$DINT := homingMethod;
	ResponseSize := 24;

	if (pRequest = NIL) | (RequestSize <> 72) then
		(pResponse + 12)^$UDINT := detailCode;
		RETURN;
	end_if;

	schemaVersion := pRequest^$UINT;
	requestFlags := (pRequest + 2)^$UINT;
	diagnosticsBuild := (pRequest + 8)^$UDINT;
	bootId := (pRequest + 12)^$UDINT;
	mapRevision := (pRequest + 16)^$UDINT;
	intent0 := (pRequest + 20)^$UDINT;
	intent1 := (pRequest + 24)^$UDINT;
	intent2 := (pRequest + 28)^$UDINT;
	intent3 := (pRequest + 32)^$UDINT;
	homePosition := (pRequest + 40)^$DINT;
	velocity := (pRequest + 44)^$DINT;
	acceleration := (pRequest + 48)^$DINT;
	distanceLimit := (pRequest + 52)^$DINT;
	torqueLimit := (pRequest + 56)^$DINT;
	bufferMode := (pRequest + 60)^$UINT;
	reservedValue := (pRequest + 62)^$UINT;
	timeoutMs := (pRequest + 64)^$UDINT;
	executeToken := (pRequest + 68)^$UDINT;
	currentBootId := GetDiagnosticsBootId();
	rawStartState := 0xFFFFFFFF;
	baseStartState := 0xFFFFFFFF;
	axisMask := 0;
	journalEligible := FALSE;
	journalPrepared := FALSE;
	preflightOnly := (AdmissionToken = 0) & (OwnerGeneration = 0);
	if (Reference >= 1) & (Reference <= 4) then
		recordBase := TO_DINT(Reference - 1) * 23;
		axisMask := TO_UDINT(1) shl TO_UDINT(Reference - 1);
		rawStartState := Ds402HomeState[recordBase]$UDINT;
		baseStartState := rawStartState and 0x00007FFF;
	end_if;
	if preflightOnly then
		// Publish the request intent before TCP may create a common reservation.
		// Stage 87 is the final publication word and can only resolve to rollback.
		if (Reference < 1) | (Reference > 4) |
			(schemaVersion <> 1) | (requestFlags <> 0) | (requestId = 0) |
			((intent0 = 0) & (intent1 = 0) & (intent2 = 0) & (intent3 = 0)) |
			(homingMethod <> 37) | (homePosition <> 0) |
			(velocity <> 0) | (acceleration <> 0) |
			(distanceLimit <> 0) | (torqueLimit <> 0) |
			(bufferMode <> 1) | (reservedValue <> 0) | (timeoutMs = 0) |
			(executeToken <> 0x32303448) then
			detailCode := 9;
		elsif diagnosticsBuild <> 1 then
			detailCode := 16;
		elsif (currentBootId = 0) | (bootId <> currentBootId) then
			detailCode := 17;
		elsif mapRevision <> LMC_DIAG_MAP_REVISION then
			detailCode := 18;
		elsif (CallerSessionEpoch = 0) | (RequestSequence = 0) |
			(sizeof(Ds402HomeState) <> 512) |
			(Ds402HomeState[92] <> 0) |
			(Ds402HomeState[109]$UDINT = 0xFFFFFFFF) then
			detailCode := 10;
		elsif (rawStartState = 2) | (rawStartState = 3) |
			(rawStartState = 4) then
			detailCode := 32;
		elsif (rawStartState <> 0) & (rawStartState <> 0x00008002) &
			(rawStartState <> 0x00008003) &
			(rawStartState <> 0x00008004) then
			detailCode := 10;
		else
			recordBase := TO_DINT(Reference - 1) * 23;
			// Slot 109 is the last committed operation generation. Intent
			// publication must not consume it.
			_memset(dest:=#Ds402HomeState[92], usByte:=0, cntr:=68);
			_memset(dest:=#Ds402HomeState[110], usByte:=0, cntr:=72);
			Ds402HomeState[93] := TO_DINT(Reference - 1);
			_memcpy(ptr1:=#Ds402HomeState[94], ptr2:=pRequest, cntr:=60);
			_memcpy(ptr1:=#Ds402HomeState[110], ptr2:=pRequest + 60,
				cntr:=12);
			Ds402HomeState[113] := CallerSessionEpoch$DINT;
			Ds402HomeState[114] := RequestSequence$DINT;
			Ds402HomeState[115] := rawStartState$DINT;
			Ds402HomeState[116]$UDINT := LMC_DIAG_DS402_INTENT_MAGIC;
			Ds402HomeState[117] := Ds402HomeState[109];
			currentCycle := ops.tAbsolute;
			if currentCycle = 0 then
				currentCycle := 1;
			end_if;
			Ds402HomeState[118] := currentCycle$DINT;
			Ds402HomeState[119] := 0;
			intentBodyCompareResult := _memcmp(ptr1:=#Ds402HomeState[94],
				ptr2:=pRequest, cntr:=60);
			intentTailCompareResult := _memcmp(ptr1:=#Ds402HomeState[110],
				ptr2:=pRequest + 60, cntr:=12);
			if (intentBodyCompareResult = 0) &
				(intentTailCompareResult = 0) &
				(Ds402HomeState[93] = TO_DINT(Reference - 1)) &
				(Ds402HomeState[113]$UDINT = CallerSessionEpoch) &
				(Ds402HomeState[114]$UDINT = RequestSequence) &
				(Ds402HomeState[115]$UDINT = rawStartState) &
				(Ds402HomeState[116]$UDINT =
				 LMC_DIAG_DS402_INTENT_MAGIC) &
				(Ds402HomeState[117] = Ds402HomeState[109]) &
				(Ds402HomeState[118] <> 0) &
				(Ds402HomeState[recordBase]$UDINT = rawStartState) then
				Ds402HomeState[92] :=
					LMC_DIAG_DS402_STAGE_RESERVE_INTENT;
				if Ds402HomeState[92] =
					LMC_DIAG_DS402_STAGE_RESERVE_INTENT then
					ResponseSize := LMC_DIAG_DS402_PREFLIGHT_READY;
					RETURN;
				end_if;
			end_if;
			detailCode := 10;
		end_if;
		(pResponse + 12)^$UDINT := detailCode;
		RETURN;
	end_if;
	intentMatches := FALSE;
	if (Reference >= 1) & (Reference <= 4) &
		(Ds402HomeState[92] = LMC_DIAG_DS402_STAGE_RESERVE_INTENT) then
		recordBase := TO_DINT(Reference - 1) * 23;
		intentBodyCompareResult := _memcmp(ptr1:=#Ds402HomeState[94],
			ptr2:=pRequest, cntr:=60);
		intentTailCompareResult := _memcmp(ptr1:=#Ds402HomeState[110],
			ptr2:=pRequest + 60, cntr:=12);
		intentMatches := (intentBodyCompareResult = 0) &
			(intentTailCompareResult = 0) &
			(Ds402HomeState[93] = TO_DINT(Reference - 1)) &
			(Ds402HomeState[113]$UDINT = CallerSessionEpoch) &
			(Ds402HomeState[114]$UDINT = RequestSequence) &
			((Ds402HomeState[115]$UDINT = 0) |
			 (Ds402HomeState[115]$UDINT = 0x00008002) |
			 (Ds402HomeState[115]$UDINT = 0x00008003) |
			 (Ds402HomeState[115]$UDINT = 0x00008004)) &
			(Ds402HomeState[116]$UDINT = LMC_DIAG_DS402_INTENT_MAGIC) &
			(Ds402HomeState[117] = Ds402HomeState[109]) &
			(Ds402HomeState[118] <> 0) &
			(Ds402HomeState[119] = 0) &
			(Ds402HomeState[120] = 0) &
			(Ds402HomeState[121] = 0) &
			(Ds402HomeState[122] = 0) &
			(Ds402HomeState[123] = 0) &
			(Ds402HomeState[124] = 0) &
			(Ds402HomeState[125] = 0) &
			(Ds402HomeState[126] = 0) &
			(Ds402HomeState[127] = 0) &
			(Ds402HomeState[recordBase]$UDINT =
			 Ds402HomeState[115]$UDINT);
	end_if;

	if (Reference < 1) | (Reference > 4) |
		(schemaVersion <> 1) | (requestFlags <> 0) | (requestId = 0) |
		((intent0 = 0) & (intent1 = 0) & (intent2 = 0) & (intent3 = 0)) |
		(homingMethod <> 37) | (homePosition <> 0) |
		(velocity <> 0) | (acceleration <> 0) |
		(distanceLimit <> 0) | (torqueLimit <> 0) |
		(bufferMode <> 1) | (reservedValue <> 0) | (timeoutMs = 0) |
		(executeToken <> 0x32303448) then
		detailCode := 9;
	elsif diagnosticsBuild <> 1 then
		detailCode := 16;
	elsif (currentBootId = 0) | (bootId <> currentBootId) then
		detailCode := 17;
	elsif mapRevision <> LMC_DIAG_MAP_REVISION then
		detailCode := 18;
	elsif (LMC_DIAG_DS402_HOME_ENABLED = FALSE) |
		(CallerSessionEpoch = 0) | (RequestSequence = 0) |
		(AdmissionToken = 0) | (OwnerGeneration = 0) |
		(IsClientConnected(#AxisOwnership) = FALSE) |
		(sizeof(Ds402HomeState) <> 512) |
		(intentMatches = FALSE) |
		(Ds402HomeState[109]$UDINT = 0xFFFFFFFF) |
		(EncoderMaintenanceState[LMC_DIAG_ENCODER_RUNTIME_BASE] <> 0) |
		(OperationState = LMC_DIAG_SDO_STATE_QUEUED) |
		(OperationState = LMC_DIAG_SDO_STATE_RUNNING) |
		(SdoInternalDrainState <> 0) then
		detailCode := 10;
	elsif (rawStartState = 2) | (rawStartState = 3) |
		(rawStartState = 4) then
		detailCode := 32;
	elsif (rawStartState <> 0) & (rawStartState <> 0x00008002) &
		(rawStartState <> 0x00008003) &
		(rawStartState <> 0x00008004) then
		detailCode := 10;
	else
		detailCode := 0;
	end_if;

	// Promote only the exact pre-reservation intent into a RESERVED rollback
	// journal. Stage 88 can only roll back; stage 89 may commit.
	journalEligible :=
		(Reference >= 1) & (Reference <= 4) &
		(schemaVersion = 1) & (requestFlags = 0) & (requestId <> 0) &
		((intent0 <> 0) | (intent1 <> 0) | (intent2 <> 0) | (intent3 <> 0)) &
		(homingMethod = 37) & (homePosition = 0) &
		(velocity = 0) & (acceleration = 0) &
		(distanceLimit = 0) & (torqueLimit = 0) &
		(bufferMode = 1) & (reservedValue = 0) & (timeoutMs <> 0) &
		(executeToken = 0x32303448) &
		(CallerSessionEpoch <> 0) & (RequestSequence <> 0) &
		(AdmissionToken <> 0) & (OwnerGeneration <> 0) &
		(sizeof(Ds402HomeState) = 512) &
		intentMatches &
		((rawStartState = 0) | (rawStartState = 0x00008002) |
		 (rawStartState = 0x00008003) | (rawStartState = 0x00008004));
	if journalEligible then
		nextGeneration := Ds402HomeState[117]$UDINT;
		if nextGeneration = 0xFFFFFFFF then
			journalEligible := FALSE;
		else
			nextGeneration += 1;
			if nextGeneration = 0 then
				journalEligible := FALSE;
			end_if;
		end_if;
	end_if;
	if journalEligible & IsClientConnected(#AxisOwnership) then
		ownerResult := AxisOwnership.ValidateAxisOwnershipIdentity(
			CommandId:=0x7D15,
			Reference:=Reference,
			ExpectedAxisMask:=axisMask,
			OwnerKind:=LMC_DIAG_OWNER_KIND_DS402_HOME,
			ResourceKind:=LMC_DIAG_RESOURCE_DS402_HOME,
			AdmissionMode:=LMC_DIAG_ADMISSION_LIFECYCLE,
			CallerSessionEpoch:=CallerSessionEpoch,
			RequestSequence:=RequestSequence,
			AdmissionToken:=AdmissionToken,
			OwnerGeneration:=OwnerGeneration,
			RequiredPhase:=LMC_DIAG_OWNER_PHASE_RESERVED,
			pIdentity:=pRequest$^void,
			IdentitySize:=RequestSize);
		if ownerResult = -1 then
			// A transient validation response still owns an exact local rollback
			// journal, but it must never progress to the commit-ready stage.
			detailCode := 10;
		elsif ownerResult <> 0 then
			journalEligible := FALSE;
		end_if;
	end_if;
	if journalEligible then
		recordBase := TO_DINT(Reference - 1) * 23;
		currentCycle := ops.tAbsolute;
		if currentCycle = 0 then
			currentCycle := 1;
		end_if;
		serviceStart := Ds402HomeState[118]$UDINT;
		if serviceStart = 0 then
			serviceStart := currentCycle;
		end_if;
		// Publish the adopted tuple before a retained tombstone can be cleared.
		// Slot 119 is the bridge commit word and is written last.
		Ds402HomeState[120] := CallerSessionEpoch$DINT;
		Ds402HomeState[121] := RequestSequence$DINT;
		Ds402HomeState[122] := AdmissionToken$DINT;
		Ds402HomeState[123] := OwnerGeneration$DINT;
		Ds402HomeState[124] := axisMask$DINT;
		Ds402HomeState[125] := LMC_DIAG_DS402_RECEIPT_PREPARED;
		Ds402HomeState[119]$UDINT := LMC_DIAG_DS402_INTENT_ADOPT_MAGIC;
		// Stage87 plus the adopted tuple remains authoritative while the selected
		// record is rebuilt. Publish state 0 as a DINT commit before byte-clearing
		// the body so a torn clear remains a replayable adopted raw intent.
		Ds402HomeState[recordBase] := 0;
		_memset(dest:=#Ds402HomeState[recordBase + 1], usByte:=0, cntr:=88);
		Ds402HomeState[recordBase + 1] := diagnosticsBuild$DINT;
		Ds402HomeState[recordBase + 2] := bootId$DINT;
		Ds402HomeState[recordBase + 3] := mapRevision$DINT;
		Ds402HomeState[recordBase + 4] := requestId$DINT;
		Ds402HomeState[recordBase + 5] := intent0$DINT;
		Ds402HomeState[recordBase + 6] := intent1$DINT;
		Ds402HomeState[recordBase + 7] := intent2$DINT;
		Ds402HomeState[recordBase + 8] := intent3$DINT;
		Ds402HomeState[recordBase + 9] := homingMethod;
		Ds402HomeState[recordBase + 10] := homePosition;
		Ds402HomeState[recordBase + 11] := velocity;
		Ds402HomeState[recordBase + 12] := acceleration;
		Ds402HomeState[recordBase + 13] := timeoutMs$DINT;
		Ds402HomeState[recordBase + 19] := currentCycle$DINT;
		Ds402HomeState[recordBase + 22] := nextGeneration$DINT;
		// Record state commits the exact body and target metadata before the WAL
		// request bytes are reused.
		Ds402HomeState[recordBase] := 1;
		_memset(dest:=#Ds402HomeState[94], usByte:=0, cntr:=60);
		_memset(dest:=#Ds402HomeState[110], usByte:=0, cntr:=36);
		_memset(dest:=#Ds402HomeState[126], usByte:=0, cntr:=8);
		Ds402HomeState[99] := nextGeneration$DINT;
		Ds402HomeState[101] := nextGeneration$DINT;
		Ds402HomeState[103] := 1;
		Ds402HomeState[105] := 8;
		Ds402HomeState[109] := nextGeneration$DINT;
		Ds402HomeState[110] := currentCycle$DINT;
		Ds402HomeState[118]$UDINT := serviceStart;
		// This publication word means rollback-only until all start gates pass.
		Ds402HomeState[92] := LMC_DIAG_DS402_STAGE_ROLLBACK_PREPARED;
		journalPrepared := TRUE;
		// Stage88 now replaces the adoption proof for the synchronous Start path.
		Ds402HomeState[119] := 0;
	elsif detailCode = 0 then
		detailCode := 10;
	end_if;
	if journalPrepared & (detailCode = 0) &
		(IsClientConnected(#AxisOwnership) = FALSE) then
		// Preserve the exact rollback-only journal across a transient owner-client
		// disconnect. The cyclic processor validates the common tuple later.
		detailCode := 10;
	end_if;

	if detailCode = 0 then
		copyResult := -1;
		if IsClientConnected(#InputLatch) then
			copyResult := InputLatch.CopySnapshot(
				pDest:=#snapshot[0], DestSize:=sizeof(snapshot));
		end_if;
		if copyResult <> 0 then
			detailCode := 10;
		else
			currentCycle := snapshot[0]$UDINT;
			serviceStart := ops.tAbsolute;
			if serviceStart = 0 then
				serviceStart := 1;
			end_if;
			healthOffset := 64 + TO_UDINT(Reference - 1) * 36;
			valueOffset := 208 + TO_UDINT(Reference - 1) * 24;
			statusWord := snapshot[TO_DINT(valueOffset + 20)]$UDINT;
			if (currentCycle = 0) | (snapshot[12]$UDINT <> 8) |
				(snapshot[16]$UDINT <> 0) |
				((snapshot[40]$UDINT and 3) <> 1) |
				(snapshot[TO_DINT(healthOffset)]$DINT = 0) |
				(snapshot[TO_DINT(healthOffset + 4)]$UDINT <> 8) |
				(snapshot[TO_DINT(healthOffset + 12)]$UDINT <> 0) |
				(snapshot[TO_DINT(healthOffset + 16)]$UDINT = 0xFFFFFFFF) |
				(snapshot[TO_DINT(healthOffset + 24)]$DINT <> 0) |
				(snapshot[TO_DINT(healthOffset + 28)]$UDINT <> currentCycle) |
				((statusWord and 0x0008) <> 0) |
				(((statusWord and 0x006F) <> 0x0040) &
				 ((statusWord and 0x006F) <> 0x0021) &
				 ((statusWord and 0x006F) <> 0x0023) &
				 ((statusWord and 0x006F) <> 0x0027)) then
				 detailCode := 10;
			else
				Ds402HomeState[recordBase + 17] := statusWord$DINT;
				Ds402HomeState[recordBase + 18] :=
					snapshot[TO_DINT(valueOffset + 12)]$DINT;
				Ds402HomeState[recordBase + 19] := currentCycle$DINT;
				Ds402HomeState[102] :=
					snapshot[TO_DINT(valueOffset + 12)]$DINT;
				Ds402HomeState[110] := currentCycle$DINT;
				Ds402HomeState[114] := statusWord$DINT;
				Ds402HomeState[115] :=
					snapshot[TO_DINT(valueOffset + 12)]$DINT;
				Ds402HomeState[118]$UDINT := serviceStart;
			end_if;
		end_if;
	end_if;

	if detailCode = 0 then
		executorConnected := FALSE;
		executorReusable := FALSE;
		case Reference of
			1:
				executorConnected := IsClientConnected(#SdoAxis1) <> 0;
				if executorConnected then
					executorReusable := SdoAxis1.IsReusable();
				end_if;
			2:
				executorConnected := IsClientConnected(#SdoAxis2) <> 0;
				if executorConnected then
					executorReusable := SdoAxis2.IsReusable();
				end_if;
			3:
				executorConnected := IsClientConnected(#SdoAxis3) <> 0;
				if executorConnected then
					executorReusable := SdoAxis3.IsReusable();
				end_if;
			4:
				executorConnected := IsClientConnected(#SdoAxis4) <> 0;
				if executorConnected then
					executorReusable := SdoAxis4.IsReusable();
				end_if;
		end_case;
		if (executorConnected = FALSE) | (executorReusable = FALSE) then
			detailCode := 10;
		end_if;
	end_if;

	if detailCode = 0 then
		if journalPrepared = FALSE then
			detailCode := 10;
		else
			// From this publication onward a warm recovery may finish Commit.
			Ds402HomeState[92] := 89;
		end_if;
	end_if;

	if (detailCode = 0) &
		(IsClientConnected(#AxisOwnership) = FALSE) then
		// Stage 89 permits warm Commit. Revoke that permission before exposing
		// the disconnect error so rejected Start cleanup remains rollback-only.
		Ds402HomeState[92] := LMC_DIAG_DS402_STAGE_ROLLBACK_PREPARED;
		detailCode := 10;
	end_if;
	if detailCode = 0 then
		ownerResult := AxisOwnership.CommitAxisOwnership(
			CommandId:=0x7D15,
			Reference:=Reference,
			ExpectedAxisMask:=axisMask,
			CallerSessionEpoch:=CallerSessionEpoch,
			RequestSequence:=RequestSequence,
			AdmissionToken:=AdmissionToken,
			OwnerGeneration:=OwnerGeneration);
		if ownerResult = 0 then
			Ds402HomeState[125] := 2;
			Ds402HomeState[92] := 1;
		else
			// A lost Commit response is accepted only after exact ACTIVE proof.
			ownerResult := AxisOwnership.ValidateAxisOwnership(
				CommandId:=0x7D15,
				Reference:=Reference,
				ExpectedAxisMask:=axisMask,
				OwnerKind:=LMC_DIAG_OWNER_KIND_DS402_HOME,
				ResourceKind:=LMC_DIAG_RESOURCE_DS402_HOME,
				AdmissionMode:=LMC_DIAG_ADMISSION_LIFECYCLE,
				CallerSessionEpoch:=CallerSessionEpoch,
				RequestSequence:=RequestSequence,
				AdmissionToken:=AdmissionToken,
				OwnerGeneration:=OwnerGeneration,
				RequiredPhase:=LMC_DIAG_OWNER_PHASE_ACTIVE);
			if ownerResult = 0 then
				Ds402HomeState[125] := 2;
				Ds402HomeState[92] := 1;
			else
				// Commit is uncertain but the handler has not run. Downgrade to the
				// rollback-only publication word before returning an error.
				Ds402HomeState[92] :=
					LMC_DIAG_DS402_STAGE_ROLLBACK_PREPARED;
				detailCode := 10;
			end_if;
		end_if;
	end_if;

	if detailCode = 0 then
		(pResponse + 4)^$UINT := 0;
		(pResponse + 6)^$INT := 0;
	end_if;
	if (detailCode <> 0) & (AdmissionToken <> 0) &
		(OwnerGeneration <> 0) & (CallerSessionEpoch <> 0) &
		(RequestSequence <> 0) then
		if (Reference >= 1) & (Reference <= 4) &
			((Ds402HomeState[92] =
			  LMC_DIAG_DS402_STAGE_ROLLBACK_PREPARED) |
			 (Ds402HomeState[92] = 89)) &
			(Ds402HomeState[93] = TO_DINT(Reference - 1)) &
			(Ds402HomeState[120]$UDINT = CallerSessionEpoch) &
			(Ds402HomeState[121]$UDINT = RequestSequence) &
			(Ds402HomeState[122]$UDINT = AdmissionToken) &
			(Ds402HomeState[123]$UDINT = OwnerGeneration) &
			(Ds402HomeState[124]$UDINT = axisMask) then
			// The local journal now owns rollback completion across task restarts.
			rollbackResult := -1;
			if IsClientConnected(#AxisOwnership) then
				rollbackResult :=
					AxisOwnership.PublishAxisOwnershipDs402Receipt(
						AxisMask:=axisMask,
						AdmissionToken:=AdmissionToken,
						OwnerGeneration:=OwnerGeneration,
						ReportKind:=LMC_DIAG_DS402_RECEIPT_ROLLBACK,
						ReportValue0:=0,
						ReportValue1:=0,
						ObservationCycle:=Ds402HomeState[110]$UDINT,
						pDs402State:=#Ds402HomeState[0],
						Ds402StateSize:=sizeof(Ds402HomeState));
			end_if;
			if rollbackResult = 0 then
				if Ds402HomeState[125] =
					LMC_DIAG_DS402_RECEIPT_PREPARED then
					Ds402HomeState[125] := 2;
				end_if;
				// Finish owner cleanup before a rejected Start response can race a
				// session-close quarantine of the still-RESERVED tuple.
				rollbackResult := -1;
				if IsClientConnected(#AxisOwnership) then
					rollbackResult :=
						AxisOwnership.PublishAxisOwnershipDs402Receipt(
							AxisMask:=axisMask,
							AdmissionToken:=AdmissionToken,
							OwnerGeneration:=OwnerGeneration,
							ReportKind:=LMC_DIAG_DS402_RECEIPT_ROLLBACK,
							ReportValue0:=0,
							ReportValue1:=0,
							ObservationCycle:=Ds402HomeState[110]$UDINT,
							pDs402State:=#Ds402HomeState[0],
							Ds402StateSize:=sizeof(Ds402HomeState));
				end_if;
				if rollbackResult = 1 then
					Ds402HomeState[92] := LMC_DIAG_DS402_STAGE_FINALIZE;
				else
					if (rollbackResult <> -1) |
						(Ds402HomeState[92] <>
						 LMC_DIAG_DS402_STAGE_ROLLBACK_PREPARED) then
						Ds402HomeState[92] := 101;
					end_if;
					detailCode := 42;
				end_if;
			elsif rollbackResult = 1 then
				Ds402HomeState[92] := LMC_DIAG_DS402_STAGE_FINALIZE;
			else
				if (rollbackResult <> -1) |
					(Ds402HomeState[92] <>
					 LMC_DIAG_DS402_STAGE_ROLLBACK_PREPARED) then
					Ds402HomeState[92] := 101;
				end_if;
				detailCode := 42;
			end_if;
		elsif Ds402HomeState[92] =
			LMC_DIAG_DS402_STAGE_RESERVE_INTENT then
			// Stage 87 has no trusted token tuple yet. Only the cyclic tokenless
			// provider may prove and resolve it; never issue a blind rollback here.
			if intentMatches = FALSE then
				Ds402HomeState[92] := 101;
			end_if;
			detailCode := 42;
		else
			// Errors before local journal publication still use exact reservation
			// rollback. No runtime record exists to recover in this branch.
			rollbackResult := -1;
			if IsClientConnected(#AxisOwnership) then
				rollbackResult := AxisOwnership.RollbackAxisOwnership(
					AdmissionToken:=AdmissionToken,
					OwnerGeneration:=OwnerGeneration,
					CallerSessionEpoch:=CallerSessionEpoch,
					RequestSequence:=RequestSequence,
					Reason:=0);
			end_if;
			if rollbackResult <> 0 then
				detailCode := 42;
			end_if;
		end_if;
	end_if;

	(pResponse + 12)^$UDINT := detailCode;

END_FUNCTION

FUNCTION LMCDiagnosticsService::HandleAxisDs402HomeOutcome
	VAR_INPUT
		Reference 	: UINT;
		pRequest 	: ^USINT;
		pResponse 	: ^USINT;
		ResponseCapacity 	: UDINT;
		CallerSessionEpoch 	: UDINT;
		RequestSize 	: UDINT;
	END_VAR
	VAR_OUTPUT
		ResponseSize 	: DINT;
	END_VAR
	VAR
		schemaVersion, requestFlags : UINT;
		requestId, diagnosticsBuild, bootId, mapRevision : UDINT;
		originalRequestId, intent0, intent1, intent2, intent3 : UDINT;
		currentBootId, detailCode, startCycle, completionCycle : UDINT;
		rawOutcomeState, baseOutcomeState : UDINT;
		homingMethod : DINT;
		recordBase : DINT;
		recordValid, outcomeStateValid : BOOL;
	END_VAR

	ResponseSize := -1;
	if (pResponse = NIL) | (ResponseCapacity < 16) then
		RETURN;
	end_if;
	_memset(dest:=pResponse, usByte:=0, cntr:=ResponseCapacity);
	pResponse^$UINT := LMC_DIAG_SCHEMA_VERSION;
	(pResponse + 4)^$UINT := 1;
	(pResponse + 6)^$INT := LMC_DIAG_ADMIN_ERROR_ID;
	detailCode := 28;
	requestId := 0;
	if (pRequest <> NIL) & (RequestSize >= 8) then
		requestId := (pRequest + 4)^$UDINT;
	end_if;
	(pResponse + 8)^$UDINT := requestId;
	ResponseSize := 16;

	if (pRequest = NIL) | (RequestSize <> 44) |
		(Reference < 1) | (Reference > 4) then
		(pResponse + 12)^$UDINT := detailCode;
		RETURN;
	end_if;

	schemaVersion := pRequest^$UINT;
	requestFlags := (pRequest + 2)^$UINT;
	diagnosticsBuild := (pRequest + 8)^$UDINT;
	bootId := (pRequest + 12)^$UDINT;
	mapRevision := (pRequest + 16)^$UDINT;
	originalRequestId := (pRequest + 20)^$UDINT;
	intent0 := (pRequest + 24)^$UDINT;
	intent1 := (pRequest + 28)^$UDINT;
	intent2 := (pRequest + 32)^$UDINT;
	intent3 := (pRequest + 36)^$UDINT;
	homingMethod := (pRequest + 40)^$DINT;
	currentBootId := GetDiagnosticsBootId();

	if (schemaVersion <> 1) | (requestFlags <> 0) | (requestId = 0) |
		(originalRequestId = 0) |
		((intent0 = 0) & (intent1 = 0) & (intent2 = 0) & (intent3 = 0)) |
		(homingMethod <> 37) then
		detailCode := 28;
	elsif diagnosticsBuild <> 1 then
		detailCode := 16;
	elsif (currentBootId = 0) | (bootId <> currentBootId) then
		detailCode := 17;
	elsif mapRevision <> LMC_DIAG_MAP_REVISION then
		detailCode := 18;
	elsif (sizeof(Ds402HomeState) <> 512) |
		(CallerSessionEpoch = 0) then
		detailCode := 29;
	else
		recordBase := TO_DINT(Reference - 1) * 23;
		rawOutcomeState := Ds402HomeState[recordBase]$UDINT;
		baseOutcomeState := rawOutcomeState and 0x00007FFF;
		outcomeStateValid :=
			(rawOutcomeState = 1) | (rawOutcomeState = 2) |
			(rawOutcomeState = 3) | (rawOutcomeState = 4) |
			(rawOutcomeState = 0x00008002) |
			(rawOutcomeState = 0x00008003) |
			(rawOutcomeState = 0x00008004);
		if rawOutcomeState = 0 then
			detailCode := 25;
		elsif outcomeStateValid = FALSE then
			detailCode := 27;
		elsif (Ds402HomeState[recordBase + 1]$UDINT <> diagnosticsBuild) |
			(Ds402HomeState[recordBase + 2]$UDINT <> bootId) |
			(Ds402HomeState[recordBase + 3]$UDINT <> mapRevision) |
			(Ds402HomeState[recordBase + 4]$UDINT <> originalRequestId) |
			(Ds402HomeState[recordBase + 5]$UDINT <> intent0) |
			(Ds402HomeState[recordBase + 6]$UDINT <> intent1) |
			(Ds402HomeState[recordBase + 7]$UDINT <> intent2) |
			(Ds402HomeState[recordBase + 8]$UDINT <> intent3) |
			(Ds402HomeState[recordBase + 9] <> homingMethod) then
			detailCode := 28;
		elsif (baseOutcomeState = 1) & (Ds402HomeState[92] = 101) &
			(Ds402HomeState[93] = TO_DINT(Reference - 1)) then
			detailCode := 26;
		else
			startCycle := Ds402HomeState[recordBase + 19]$UDINT;
			completionCycle := Ds402HomeState[recordBase + 20]$UDINT;
			recordValid := (startCycle <> 0) &
				(Ds402HomeState[recordBase + 22]$UDINT <> 0);
			if baseOutcomeState = 1 then
				recordValid := recordValid & (completionCycle = 0) &
					(Ds402HomeState[recordBase + 14] = 0) &
					(Ds402HomeState[recordBase + 15] = 0) &
					(Ds402HomeState[recordBase + 16] = 0) &
					(Ds402HomeState[recordBase + 21] = 0);
			elsif baseOutcomeState = 2 then
				recordValid := recordValid & (completionCycle >= startCycle) &
					(Ds402HomeState[recordBase + 14] = 0) &
					(Ds402HomeState[recordBase + 15] = 0) &
					(Ds402HomeState[recordBase + 16] = 0) &
					(Ds402HomeState[recordBase + 21] = 0) &
					(Ds402HomeState[recordBase + 18] = 0) &
					((Ds402HomeState[recordBase + 17]$UDINT and
					  0x0008) = 0) &
					((Ds402HomeState[recordBase + 17]$UDINT and
					  0x2000) = 0) &
					(((Ds402HomeState[recordBase + 17]$UDINT and
					   0x006F) = 0x0040) |
					 ((Ds402HomeState[recordBase + 17]$UDINT and
					   0x006F) = 0x0021) |
					 ((Ds402HomeState[recordBase + 17]$UDINT and
					   0x006F) = 0x0023) |
					 ((Ds402HomeState[recordBase + 17]$UDINT and
					   0x006F) = 0x0027));
			elsif baseOutcomeState = 3 then
				recordValid := recordValid & (completionCycle >= startCycle) &
					(Ds402HomeState[recordBase + 14] = 1) &
					(((Ds402HomeState[recordBase + 16] = 11) &
					  (Ds402HomeState[recordBase + 15] = -6) &
					  (Ds402HomeState[recordBase + 21] <> 0)) |
					 ((Ds402HomeState[recordBase + 16] = 10) &
					  (Ds402HomeState[recordBase + 15] = LMC_DIAG_ADMIN_ERROR_ID) &
					  (Ds402HomeState[recordBase + 21] = 0)) |
					 ((Ds402HomeState[recordBase + 16] = 30) &
					  (Ds402HomeState[recordBase + 15] = LMC_DIAG_ADMIN_ERROR_ID)));
			elsif baseOutcomeState = 4 then
				recordValid := recordValid & (completionCycle >= startCycle) &
					(Ds402HomeState[recordBase + 14] = 1) &
					(Ds402HomeState[recordBase + 15] = LMC_DIAG_ADMIN_ERROR_ID) &
					(Ds402HomeState[recordBase + 16] = 31) &
					(Ds402HomeState[recordBase + 21] = 0);
			else
				recordValid := FALSE;
			end_if;
			if recordValid then
				detailCode := 0;
			else
				detailCode := 27;
			end_if;
		end_if;
	end_if;

	if detailCode <> 0 then
		(pResponse + 12)^$UDINT := detailCode;
		RETURN;
	end_if;
	if ResponseCapacity < 92 then
		ResponseSize := -1;
		RETURN;
	end_if;

	(pResponse + 4)^$UINT := 0;
	(pResponse + 6)^$INT := 0;
	(pResponse + 12)^$UDINT := 0;
	(pResponse + 16)^$UINT := baseOutcomeState$UINT;
	(pResponse + 20)^$UDINT := Ds402HomeState[recordBase + 1]$UDINT;
	(pResponse + 24)^$UDINT := Ds402HomeState[recordBase + 2]$UDINT;
	(pResponse + 28)^$UDINT := Ds402HomeState[recordBase + 3]$UDINT;
	(pResponse + 32)^$UDINT := Ds402HomeState[recordBase + 4]$UDINT;
	(pResponse + 36)^$UDINT := Ds402HomeState[recordBase + 5]$UDINT;
	(pResponse + 40)^$UDINT := Ds402HomeState[recordBase + 6]$UDINT;
	(pResponse + 44)^$UDINT := Ds402HomeState[recordBase + 7]$UDINT;
	(pResponse + 48)^$UDINT := Ds402HomeState[recordBase + 8]$UDINT;
	(pResponse + 52)^$UINT := Reference;
	(pResponse + 56)^$DINT := Ds402HomeState[recordBase + 9];
	(pResponse + 60)^$UINT := Ds402HomeState[recordBase + 14]$UINT;
	(pResponse + 62)^$INT := Ds402HomeState[recordBase + 15]$INT;
	(pResponse + 64)^$UDINT := Ds402HomeState[recordBase + 16]$UDINT;
	(pResponse + 68)^$UINT := Ds402HomeState[recordBase + 17]$UINT;
	(pResponse + 72)^$DINT := Ds402HomeState[recordBase + 18];
	(pResponse + 76)^$UDINT := Ds402HomeState[recordBase + 19]$UDINT;
	(pResponse + 80)^$UDINT := Ds402HomeState[recordBase + 20]$UDINT;
	(pResponse + 84)^$UDINT := Ds402HomeState[recordBase + 21]$UDINT;
	(pResponse + 88)^$UDINT := Ds402HomeState[recordBase + 22]$UDINT;
	ResponseSize := 92;

END_FUNCTION

FUNCTION LMCDiagnosticsService::HandleAxisDs402HomeRetire
	VAR_INPUT
		Reference 	: UINT;
		pRequest 	: ^USINT;
		pResponse 	: ^USINT;
		ResponseCapacity 	: UDINT;
		CallerSessionEpoch 	: UDINT;
		RequestSize 	: UDINT;
	END_VAR
	VAR_OUTPUT
		ResponseSize 	: DINT;
	END_VAR
	VAR
		schemaVersion, requestFlags : UINT;
		requestId, diagnosticsBuild, bootId, mapRevision : UDINT;
		originalRequestId, intent0, intent1, intent2, intent3 : UDINT;
		recordGeneration, detailCode, currentBootId : UDINT;
		rawRetireState, baseRetireState : UDINT;
		homingMethod, recordBase : DINT;
		retireStateValid : BOOL;
	END_VAR

	ResponseSize := -1;
	if (pResponse = NIL) | (ResponseCapacity < 16) then
		RETURN;
	end_if;
	_memset(dest:=pResponse, usByte:=0, cntr:=ResponseCapacity);
	pResponse^$UINT := LMC_DIAG_SCHEMA_VERSION;
	(pResponse + 4)^$UINT := 1;
	(pResponse + 6)^$INT := LMC_DIAG_ADMIN_ERROR_ID;
	requestId := 0;
	if (pRequest <> NIL) & (RequestSize >= 8) then
		requestId := (pRequest + 4)^$UDINT;
	end_if;
	(pResponse + 8)^$UDINT := requestId;
	ResponseSize := 16;
	detailCode := 28;
	if (pRequest = NIL) | (RequestSize <> 48) |
		(Reference < 1) | (Reference > 4) then
		(pResponse + 12)^$UDINT := detailCode;
		RETURN;
	end_if;

	schemaVersion := pRequest^$UINT;
	requestFlags := (pRequest + 2)^$UINT;
	requestId := (pRequest + 4)^$UDINT;
	diagnosticsBuild := (pRequest + 8)^$UDINT;
	bootId := (pRequest + 12)^$UDINT;
	mapRevision := (pRequest + 16)^$UDINT;
	originalRequestId := (pRequest + 20)^$UDINT;
	intent0 := (pRequest + 24)^$UDINT;
	intent1 := (pRequest + 28)^$UDINT;
	intent2 := (pRequest + 32)^$UDINT;
	intent3 := (pRequest + 36)^$UDINT;
	homingMethod := (pRequest + 40)^$DINT;
	recordGeneration := (pRequest + 44)^$UDINT;
	currentBootId := GetDiagnosticsBootId();

	if (schemaVersion <> 1) | (requestFlags <> 0) | (requestId = 0) |
		(originalRequestId = 0) | (recordGeneration = 0) |
		((intent0 = 0) & (intent1 = 0) & (intent2 = 0) & (intent3 = 0)) |
		(homingMethod <> 37) then
		detailCode := 28;
	elsif diagnosticsBuild <> 1 then
		detailCode := 16;
	elsif (currentBootId = 0) | (bootId <> currentBootId) then
		detailCode := 17;
	elsif mapRevision <> LMC_DIAG_MAP_REVISION then
		detailCode := 18;
	elsif (sizeof(Ds402HomeState) <> 512) |
		(CallerSessionEpoch = 0) then
		detailCode := 29;
	else
		recordBase := TO_DINT(Reference - 1) * 23;
		rawRetireState := Ds402HomeState[recordBase]$UDINT;
		baseRetireState := rawRetireState and 0x00007FFF;
		retireStateValid :=
			(rawRetireState = 2) | (rawRetireState = 3) |
			(rawRetireState = 4) | (rawRetireState = 0x00008002) |
			(rawRetireState = 0x00008003) |
			(rawRetireState = 0x00008004);
		if rawRetireState = 0 then
			detailCode := 25;
		elsif rawRetireState = 1 then
			detailCode := 26;
		elsif retireStateValid = FALSE then
			detailCode := 27;
		elsif (Ds402HomeState[recordBase + 1]$UDINT <> diagnosticsBuild) |
			(Ds402HomeState[recordBase + 2]$UDINT <> bootId) |
			(Ds402HomeState[recordBase + 3]$UDINT <> mapRevision) |
			(Ds402HomeState[recordBase + 4]$UDINT <> originalRequestId) |
			(Ds402HomeState[recordBase + 5]$UDINT <> intent0) |
			(Ds402HomeState[recordBase + 6]$UDINT <> intent1) |
			(Ds402HomeState[recordBase + 7]$UDINT <> intent2) |
			(Ds402HomeState[recordBase + 8]$UDINT <> intent3) |
			(Ds402HomeState[recordBase + 9] <> homingMethod) |
			(Ds402HomeState[recordBase + 22]$UDINT <> recordGeneration) then
			detailCode := 28;
		else
			detailCode := 0;
		end_if;
	end_if;

	if detailCode = 0 then
		ResponseSize := HandleAxisDs402HomeOutcome(
			Reference:=Reference, pRequest:=pRequest, pResponse:=pResponse,
			ResponseCapacity:=ResponseCapacity,
			CallerSessionEpoch:=CallerSessionEpoch, RequestSize:=44);
		if ResponseSize <> 92 then
			RETURN;
		end_if;
		if (pResponse + 88)^$UDINT <> recordGeneration then
			detailCode := 28;
		end_if;
		if detailCode = 0 then
			if rawRetireState = baseRetireState then
				Ds402HomeState[recordBase] :=
					TO_DINT(baseRetireState or 0x00008000);
			end_if;
		end_if;
	end_if;
	if detailCode <> 0 then
		(pResponse + 4)^$UINT := 1;
		(pResponse + 6)^$INT := LMC_DIAG_ADMIN_ERROR_ID;
		(pResponse + 12)^$UDINT := detailCode;
		ResponseSize := 16;
	end_if;

END_FUNCTION

FUNCTION LMCDiagnosticsService::ProcessAxisDs402Home
	VAR
		snapshot : ARRAY [0..303] OF USINT;
		preemptionSnapshot : ARRAY [0..215] OF USINT;
		completion : LMCSdoExecutor::LMCSdoExecutorResult;
		stage, nextStage, activeIndex, recordBase : DINT;
		axisReference, preemptionCleanupKind : UINT;
		currentCycle, previousCycle, startCycle, elapsedCycles : UDINT;
		serviceNow, serviceStart, cleanupStart : UDINT;
		timeoutMs, remainingMs, healthOffset, valueOffset : UDINT;
		statusWord, baseState, sdoToken, sdoData, failureDetail, failureNative : UDINT;
		axisMask, admissionToken, ownerGeneration : UDINT;
		ds402ProcessOwnerSessionEpoch, ownerRequestSequence : UDINT;
		safetyAdmissionToken, safetyOwnerGeneration : UDINT;
		sdoIndex, sdoLength : UINT;
		homeSdoSubIndex : USINT;
		actualPosition : DINT;
		copyResult, completionResult, mailboxResult, orphanResult : DINT;
		preemptionResult : DINT;
		ownerResult : DINT;
		receiptResult : DINT;
		receiptKind : DINT;
		receiptPhase : DINT;
		receiptGeneration : UDINT;
		terminalRecordState : DINT;
		startResult : iprStates;
		snapshotValid, newCycle, executorConnected, executorReusable : BOOL;
		startSdo, waitSdo, sdoIsWrite, failure : BOOL;
		preemptionSnapshotValid, preemptionCleanup, cleanupExpired : BOOL;
	END_VAR

	stage := Ds402HomeState[92];
	receiptResult := HandleAxisDs402HomeReceiptStages(Stage:=stage);
	if receiptResult <> 0 then
		RETURN;
	end_if;
	activeIndex := Ds402HomeState[93];
	admissionToken := Ds402HomeState[122]$UDINT;
	ownerGeneration := Ds402HomeState[123]$UDINT;
	_memset(dest:=#preemptionSnapshot[0], usByte:=0,
		cntr:=sizeof(preemptionSnapshot));
	preemptionResult := -1;
	if IsClientConnected(#AxisOwnership) & (admissionToken <> 0) &
		(ownerGeneration <> 0) then
		preemptionResult := AxisOwnership.CopyAxisOwnershipPreemption(
			PreemptedAdmissionToken:=admissionToken,
			PreemptedOwnerGeneration:=ownerGeneration,
			pDest:=#preemptionSnapshot[0],
			DestSize:=sizeof(preemptionSnapshot));
	end_if;
	if preemptionResult = LMC_DIAG_PREEMPT_PENDING_FREEZE then
		// A RESERVED safety owner may freeze any normal stage for at most one
		// second from the DS402 service start; neither owner is mutated here.
		serviceStart := Ds402HomeState[118]$UDINT;
		cleanupExpired := (serviceStart <> 0) &
			((ops.tAbsolute - serviceStart) >= 1000);
		if cleanupExpired then
			Ds402HomeState[92] := 101;
		end_if;
		RETURN;
	end_if;
	if (preemptionResult < 0) |
		(preemptionResult > LMC_DIAG_PREEMPT_CLEANUP_QUARANTINED) then
		Ds402HomeState[92] := 101;
		RETURN;
	end_if;
	if (activeIndex < 0) | (activeIndex > 3) |
		(sizeof(Ds402HomeState) <> 512) then
		Ds402HomeState[92] := 101;
		RETURN;
	end_if;

	axisReference := TO_UINT(activeIndex + 1);
	recordBase := activeIndex * 23;
	axisMask := Ds402HomeState[124]$UDINT;
	ds402ProcessOwnerSessionEpoch := Ds402HomeState[120]$UDINT;
	ownerRequestSequence := Ds402HomeState[121]$UDINT;
	if (axisMask <> (TO_UDINT(1) shl TO_UDINT(activeIndex))) |
		(ds402ProcessOwnerSessionEpoch = 0) | (ownerRequestSequence = 0) |
		(admissionToken = 0) | (ownerGeneration = 0) |
		(Ds402HomeState[125] <> 2) then
		Ds402HomeState[92] := 101;
		RETURN;
	end_if;
	serviceNow := ops.tAbsolute;
	serviceStart := Ds402HomeState[118]$UDINT;
	cleanupStart := Ds402HomeState[119]$UDINT;
	currentCycle := Ds402HomeState[110]$UDINT;
	previousCycle := currentCycle;
	statusWord := Ds402HomeState[114]$UDINT;
	actualPosition := Ds402HomeState[115];
	preemptionCleanup := FALSE;
	if preemptionResult <> 0 then
		preemptionSnapshotValid :=
			(preemptionSnapshot[0]$UDINT =
			 LMC_DIAG_PREEMPT_SNAPSHOT_MAGIC) &
			(preemptionSnapshot[4]$UDINT =
			 LMC_DIAG_PREEMPT_SNAPSHOT_VERSION) &
			(preemptionSnapshot[8]$UDINT =
			 LMC_DIAG_PREEMPT_SNAPSHOT_HEADER_SIZE) &
			(preemptionSnapshot[12]$UDINT =
			 LMC_DIAG_PREEMPT_SNAPSHOT_TOTAL_SIZE) &
			(preemptionSnapshot[16]$DINT = preemptionResult) &
			(preemptionSnapshot[32]$UDINT = axisMask) &
			(preemptionSnapshot[36]$UDINT = admissionToken) &
			(preemptionSnapshot[40]$UDINT = ownerGeneration) &
			(preemptionSnapshot[44]$UDINT =
			 ds402ProcessOwnerSessionEpoch) &
			(preemptionSnapshot[48]$UDINT = ownerRequestSequence) &
			(preemptionSnapshot[52]$UDINT = 0x7D15) &
			(preemptionSnapshot[56]$UDINT = TO_UDINT(axisReference)) &
			(preemptionSnapshot[60]$UDINT =
			 LMC_DIAG_OWNER_KIND_DS402_HOME) &
			(preemptionSnapshot[64]$UDINT =
			 LMC_DIAG_RESOURCE_DS402_HOME) &
			(preemptionSnapshot[68]$UDINT =
			 LMC_DIAG_ADMISSION_LIFECYCLE) &
			(Ds402HomeState[recordBase] = 1) &
			(Ds402HomeState[101]$UDINT <> 0) &
			(((stage >= 1) & (stage <= 34)) |
			 ((stage >= 90) & (stage <= 101))) &
			(preemptionSnapshot[72]$UDINT =
			 LMC_DIAG_OWNER_STATE_DS402_HOME_ACTIVE) &
			(preemptionSnapshot[76]$UDINT = 72) &
			((preemptionSnapshot[104]$UDINT and axisMask) = axisMask) &
			(preemptionSnapshot[108]$UDINT <> 0) &
			(preemptionSnapshot[112]$UDINT <> 0) &
			((preemptionSnapshot[124]$UDINT =
			  LMC_DIAG_OWNER_STATE_SAFETY_PREEMPTING) |
			 (preemptionSnapshot[124]$UDINT =
			  LMC_DIAG_OWNER_STATE_QUARANTINED)) &
			(preemptionSnapshot[136]$UDINT =
			 LMC_DIAG_ADMISSION_SAFETY) &
			(preemptionSnapshot[144]$UINT = LMC_DIAG_SCHEMA_VERSION) &
			(preemptionSnapshot[146]$UINT = 0) &
			(preemptionSnapshot[148]$UDINT =
			 Ds402HomeState[recordBase + 4]$UDINT) &
			(preemptionSnapshot[152]$UDINT =
			 Ds402HomeState[recordBase + 1]$UDINT) &
			(preemptionSnapshot[156]$UDINT =
			 Ds402HomeState[recordBase + 2]$UDINT) &
			(preemptionSnapshot[160]$UDINT =
			 Ds402HomeState[recordBase + 3]$UDINT) &
			(preemptionSnapshot[164]$UDINT =
			 Ds402HomeState[recordBase + 5]$UDINT) &
			(preemptionSnapshot[168]$UDINT =
			 Ds402HomeState[recordBase + 6]$UDINT) &
			(preemptionSnapshot[172]$UDINT =
			 Ds402HomeState[recordBase + 7]$UDINT) &
			(preemptionSnapshot[176]$UDINT =
			 Ds402HomeState[recordBase + 8]$UDINT) &
			(preemptionSnapshot[180]$DINT =
			 Ds402HomeState[recordBase + 9]) &
			(preemptionSnapshot[184]$DINT =
			 Ds402HomeState[recordBase + 10]) &
			(preemptionSnapshot[188]$DINT =
			 Ds402HomeState[recordBase + 11]) &
			(preemptionSnapshot[192]$DINT =
			 Ds402HomeState[recordBase + 12]) &
			(preemptionSnapshot[196]$DINT = 0) &
			(preemptionSnapshot[200]$DINT = 0) &
			(preemptionSnapshot[204]$UINT = 1) &
			(preemptionSnapshot[206]$UINT = 0) &
			(preemptionSnapshot[208]$UDINT =
			 Ds402HomeState[recordBase + 13]$UDINT) &
			(preemptionSnapshot[212]$UDINT = 0x32303448);
		if preemptionResult = LMC_DIAG_PREEMPT_CLEANUP_REQUIRED then
			preemptionSnapshotValid := preemptionSnapshotValid &
				((preemptionSnapshot[24]$UDINT and axisMask) = axisMask) &
				((preemptionSnapshot[28]$UDINT and axisMask) = 0) &
				(preemptionSnapshot[124]$UDINT <>
				 LMC_DIAG_OWNER_STATE_RESERVED);
		elsif preemptionResult = LMC_DIAG_PREEMPT_CLEANUP_COMPLETE then
			preemptionSnapshotValid := preemptionSnapshotValid &
				((preemptionSnapshot[28]$UDINT and axisMask) = axisMask);
		end_if;
		if preemptionSnapshotValid = FALSE then
			Ds402HomeState[92] := 101;
			RETURN;
		end_if;
		if preemptionResult = LMC_DIAG_PREEMPT_CLEANUP_COMPLETE then
			if currentCycle < Ds402HomeState[recordBase + 19]$UDINT then
				currentCycle := Ds402HomeState[recordBase + 19]$UDINT;
			end_if;
			Ds402HomeState[recordBase + 14] := 1;
			Ds402HomeState[recordBase + 15] := LMC_DIAG_ADMIN_ERROR_ID;
			Ds402HomeState[recordBase + 16] := 31;
			Ds402HomeState[recordBase + 20] := currentCycle$DINT;
			Ds402HomeState[recordBase + 21] := 0;
			Ds402HomeState[101] := 0;
			Ds402HomeState[recordBase] := 4;
			Ds402HomeState[92] := 0;
			RETURN;
		elsif preemptionResult =
			LMC_DIAG_PREEMPT_CLEANUP_QUARANTINED then
			Ds402HomeState[92] := 101;
			RETURN;
		end_if;
		safetyAdmissionToken := preemptionSnapshot[108]$UDINT;
		safetyOwnerGeneration := preemptionSnapshot[112]$UDINT;
		preemptionCleanup := TRUE;
	end_if;
	snapshotValid := FALSE;
	newCycle := FALSE;
	copyResult := -1;
	if IsClientConnected(#InputLatch) then
		copyResult := InputLatch.CopySnapshot(
			pDest:=#snapshot[0], DestSize:=sizeof(snapshot));
	end_if;
	if (copyResult = 0) & (snapshot[0]$UDINT <> 0) then
		snapshotValid := TRUE;
		currentCycle := snapshot[0]$UDINT;
		newCycle := currentCycle <> previousCycle;
		healthOffset := 64 + TO_UDINT(activeIndex) * 36;
		valueOffset := 208 + TO_UDINT(activeIndex) * 24;
		statusWord := snapshot[TO_DINT(valueOffset + 20)]$UDINT;
		baseState := statusWord and 0x006F;
		actualPosition := snapshot[TO_DINT(valueOffset + 12)]$DINT;
		Ds402HomeState[recordBase + 17] := statusWord$DINT;
		Ds402HomeState[recordBase + 18] := actualPosition;
		Ds402HomeState[114] := statusWord$DINT;
		Ds402HomeState[115] := actualPosition;
		if newCycle then
			Ds402HomeState[110] := currentCycle$DINT;
		end_if;
	end_if;

	failure := FALSE;
	failureDetail := 30;
	failureNative := 0;
	if preemptionCleanup & (stage < 90) then
		// Skip every normal Home transition and enter only owner cleanup.
		failure := TRUE;
		failureDetail := 31;
		failureNative := preemptionSnapshot[116]$UDINT;
	elsif stage < 90 then
		if LMC_DIAG_DS402_HOME_ENABLED = FALSE then
			failure := TRUE;
			failureNative := 10;
		elsif (Ds402HomeState[recordBase] <> 1) |
			(Ds402HomeState[recordBase + 2]$UDINT <> GetDiagnosticsBootId()) |
			(Ds402HomeState[recordBase + 3]$UDINT <> LMC_DIAG_MAP_REVISION) then
			failure := TRUE;
			failureNative := 17;
		elsif snapshotValid = FALSE then
			failure := TRUE;
			failureNative := 11;
		elsif (snapshot[12]$UDINT <> 8) | (snapshot[16]$UDINT <> 0) |
			((snapshot[40]$UDINT and 3) <> 1) |
			(snapshot[TO_DINT(healthOffset)]$DINT = 0) |
			(snapshot[TO_DINT(healthOffset + 4)]$UDINT <> 8) |
			(snapshot[TO_DINT(healthOffset + 12)]$UDINT <> 0) |
			(snapshot[TO_DINT(healthOffset + 16)]$UDINT = 0xFFFFFFFF) |
			(snapshot[TO_DINT(healthOffset + 24)]$DINT <> 0) |
			(snapshot[TO_DINT(healthOffset + 28)]$UDINT <> currentCycle) |
			((statusWord and 0x0008) <> 0) |
			((baseState <> 0x0040) & (baseState <> 0x0021) &
			 (baseState <> 0x0023) & (baseState <> 0x0027)) then
			failure := TRUE;
			failureNative := 19;
		end_if;
		startCycle := Ds402HomeState[recordBase + 19]$UDINT;
		timeoutMs := Ds402HomeState[recordBase + 13]$UDINT;
		if (serviceNow - serviceStart) >= timeoutMs then
			failure := TRUE;
			failureNative := LMC_DIAG_SDO_ABORT_TIMEOUT;
		end_if;
	end_if;

	if (failure = FALSE) & (stage < 90) then
		case stage of
			1:
				if newCycle then
					if ((statusWord and 0x0008) <> 0) |
						((baseState <> 0x0040) & (baseState <> 0x0021) &
						 (baseState <> 0x0023) & (baseState <> 0x0027)) then
						failure := TRUE;
						failureNative := 10;
					elsif actualPosition = Ds402HomeState[102] then
						Ds402HomeState[103] += 1;
					else
						Ds402HomeState[102] := actualPosition;
						Ds402HomeState[103] := 1;
					end_if;
					if Ds402HomeState[103] >= 3 then
						Ds402HomeState[92] := 2;
					end_if;
				end_if;

			14:
				mailboxResult := InputLatch.SubmitDs402HomeControl(
					OperationToken:=Ds402HomeState[101]$UDINT,
					AxisReference:=axisReference, Command:=1);
				if mailboxResult = 0 then
					// Runtime slot 117 means the RT control-word owner may be held.
					Ds402HomeState[117] := 1;
					Ds402HomeState[92] := 16;
				elsif mailboxResult = 1 then
					Ds402HomeState[117] := 1;
					Ds402HomeState[92] := 15;
				else
					failure := TRUE;
					failureDetail := 11;
					failureNative := TO_UDINT(0 - mailboxResult);
				end_if;

			15:
				mailboxResult := InputLatch.GetDs402HomeControlState(
					OperationToken:=Ds402HomeState[101]$UDINT);
				if mailboxResult = 0 then
					Ds402HomeState[117] := 1;
					Ds402HomeState[92] := 16;
				elsif mailboxResult <> 1 then
					failure := TRUE;
					failureDetail := 11;
					failureNative := TO_UDINT(0 - mailboxResult);
				end_if;

			20:
				if newCycle then
					if (statusWord and 0x3000) = 0 then
						Ds402HomeState[111] := 1;
						Ds402HomeState[92] := 21;
					else
						failure := TRUE;
						failureNative := statusWord;
					end_if;
				end_if;

			21:
				mailboxResult := InputLatch.SubmitDs402HomeControl(
					OperationToken:=Ds402HomeState[101]$UDINT,
					AxisReference:=axisReference, Command:=2);
				if mailboxResult = 0 then
					Ds402HomeState[104] := currentCycle$DINT;
					Ds402HomeState[102] := actualPosition;
					Ds402HomeState[103] := 0;
					Ds402HomeState[92] := 23;
				elsif mailboxResult = 1 then
					// Once SetHigh is queued, the drive coordinate may change before
					// its result is observed. Cleanup must therefore require alignment.
					Ds402HomeState[104] := currentCycle$DINT;
					Ds402HomeState[102] := actualPosition;
					Ds402HomeState[103] := 0;
					Ds402HomeState[92] := 22;
				else
					failure := TRUE;
					failureDetail := 11;
					failureNative := TO_UDINT(0 - mailboxResult);
				end_if;

			22:
				mailboxResult := InputLatch.GetDs402HomeControlState(
					OperationToken:=Ds402HomeState[101]$UDINT);
				if mailboxResult = 0 then
					Ds402HomeState[104] := currentCycle$DINT;
					Ds402HomeState[92] := 23;
				elsif mailboxResult <> 1 then
					failure := TRUE;
					failureDetail := 11;
					failureNative := TO_UDINT(0 - mailboxResult);
				end_if;

			23:
				if newCycle then
					if (statusWord and 0x2000) <> 0 then
						failure := TRUE;
						failureNative := statusWord;
					elsif (Ds402HomeState[111] <> 0) &
						((statusWord and 0x1000) <> 0) &
						((statusWord and 0x0400) <> 0) then
						if actualPosition = Ds402HomeState[recordBase + 10] then
							if actualPosition = Ds402HomeState[102] then
								Ds402HomeState[103] += 1;
							else
								Ds402HomeState[102] := actualPosition;
								Ds402HomeState[103] := 1;
							end_if;
							if Ds402HomeState[103] >= 3 then
								Ds402HomeState[92] := 24;
							end_if;
						else
							Ds402HomeState[103] := 0;
						end_if;
					else
						Ds402HomeState[103] := 0;
					end_if;
				end_if;

			24:
				mailboxResult := InputLatch.SubmitDs402HomeControl(
					OperationToken:=Ds402HomeState[101]$UDINT,
					AxisReference:=axisReference, Command:=3);
				if mailboxResult = 0 then
					Ds402HomeState[92] := 26;
				elsif mailboxResult = 1 then
					Ds402HomeState[92] := 25;
				else
					failure := TRUE;
					failureDetail := 11;
					failureNative := TO_UDINT(0 - mailboxResult);
				end_if;

			25:
				mailboxResult := InputLatch.GetDs402HomeControlState(
					OperationToken:=Ds402HomeState[101]$UDINT);
				if mailboxResult = 0 then
					Ds402HomeState[92] := 26;
				elsif mailboxResult <> 1 then
					failure := TRUE;
					failureDetail := 11;
					failureNative := TO_UDINT(0 - mailboxResult);
				end_if;

			26:
				mailboxResult := InputLatch.SubmitDs402HomeSetpointAlignment(
					OperationToken:=Ds402HomeState[101]$UDINT,
					AxisReference:=axisReference,
					ActualPosition:=actualPosition);
				if mailboxResult = 0 then
					Ds402HomeState[92] := 28;
				elsif mailboxResult = 1 then
					Ds402HomeState[92] := 27;
				else
					failure := TRUE;
					failureDetail := 11;
					failureNative := TO_UDINT(0 - mailboxResult);
				end_if;

			27:
				mailboxResult := InputLatch.GetDs402HomeControlState(
					OperationToken:=Ds402HomeState[101]$UDINT);
				if mailboxResult = 0 then
					Ds402HomeState[92] := 28;
				elsif mailboxResult <> 1 then
					failure := TRUE;
					failureDetail := 11;
					failureNative := TO_UDINT(0 - mailboxResult);
				end_if;
